
// ===== library types =====

TYPE "mettlerToledoInd560Udt"
   STRUCT
      readMsgSlot : Array[1..4] of Struct
         cmdRespons : Struct
            FP_1 : Bool;
            FP_2 : Bool;
            FP_3 : Bool;
            FP_4 : Bool;
            FP_5 : Bool;
            data_integrity : Bool;
            cmdAck1 : Bool;
            cmdAck2 : Bool;
         END_STRUCT;
         reserved : Byte;   // volt
         data : Real;
         scale_status : Struct
            x08_Enter_Key : Bool;
            x09_Input_1 : Bool;
            x10_Input_2 : Bool;
            x11_Input_3 : Bool;
            x12_Motion : Bool;
            x13_Net_Mode : Bool;
            x14_Data_Integrity_2 : Bool;
            x15_Data_OK : Bool;
            x00_Target_1 : Bool;
            x01_Comparator_1 : Bool;
            x02_Targe_2 : Bool;
            x03_Comparator_2 : Bool;
            x04_Target_3 : Bool;
            x05_Alway_true : Bool;
            x06_TE_bit_1 : Bool;
            x07_TE_bit_2 : Bool;
         END_STRUCT;
      END_STRUCT;
      writeMsgSlot : Array[1..4] of Struct
         cmd : UInt;
         data : Real;
      END_STRUCT;
      run : Struct   // Data calculated from readMsgSlot
         PF : Array[1..4] of USInt;   // Floating point input indication
         cmdAck : Array[1..4] of USInt;
      END_STRUCT;
      occupiedMsgSlots : Array[1..4] of Bool;
      queryDone : Struct
         read : Bool;
         write : Bool;
      END_STRUCT;
   END_STRUCT;
END_TYPE

// folder: Library/Modbus/Core/sb

TYPE "mb_station_block_udt"
   STRUCT
      conf : Struct   // Configuration
         disable : Bool;   // Skip all queries
         read_only : Bool;   // Skip all write queries. (fc 5,6,15,16)
         max_comm_error : USInt := 2;   // Repeating erros before communication_error flag is set
         exec_x_quries : USInt := 1;   // Number of queries to be exec. at each loop.
      END_STRUCT;
      out : Struct   // Outputs
         error : Bool;   // All errors, including communication errors
         error_comm : Bool;   // only communication errors
         finnish : Bool;   // qid is handed over to next device.
      END_STRUCT;
      log : Struct   // Logging for development and debugging.
         connected_time : DTL;   // The time the device was connected to the bus
         disconnected_time : DTL;   // The time, if a device was disconnected to the bus
         done_cnt : UDInt;   // Successfully queries counter for this device
         error_comm_cnt : UDInt;   // Communication erros cnt.
         error_exception_cnt : UDInt;   // Failed queries counter for this device
         error_status : Word;   // Status code from mb_master or mb_client
         error_data_addr : UDInt;   // d_addr for last failed querie; handy for troubleshooting
      END_STRUCT;
      z : Struct   // Internal states.
         header_qid : UInt;   // qid value at device header
         comm_err_cnt : USInt;   // Repeating communication errors
         exec_cnt : USInt;   // Numb. of exec. q. this loop
         offset_qid : UInt := 1;   // Device query id.
         err_hold : Bool;   // Help var for .out.error
      END_STRUCT;
   END_STRUCT;
END_TYPE

// folder: (top level)

FUNCTION_BLOCK "modbus_test"   // FB3, SCL
{ S7_Optimized_Access := 'TRUE' }
VERSION : 0.1
   VAR
      mb_query : "mb_query";
      mb_master_1200_ctrl : "mb_master_1200_ctrl";
      temperature_1 : "Jdrk_RS_WS_N01_8";
      temperature_2 : "Jdrk_RS_WS_N01_8";
      temperature_3 : "Jdrk_RS_WS_N01_8";
      sb_temp_no_answer_1 : "sb_temp_no_anser";
      sb_temp_no_answer_2 : "sb_temp_no_anser";
      sb_temp_no_answer_3 : "sb_temp_no_anser";
      sb_temp_error_1 : "sb_temp_error";
      sb_temp_error_2 : "sb_temp_error";
      sb_temp_error_3 : "sb_temp_error";
   END_VAR
BEGIN
   #mb_master_1200_ctrl.conf.parity := 0;
   #mb_master_1200_ctrl(hardware_id := 263, // "Local~CB_1241_(RS485)",
                        baud := 9600,
                        mb_query := #mb_query);

   #temperature_1(mb_query := #mb_query);
   #temperature_2(mb_query := #mb_query);
   #temperature_3(mb_query := #mb_query);

   #sb_temp_no_answer_1(mb_query := #mb_query);
   #sb_temp_no_answer_2(mb_query := #mb_query);
   #sb_temp_no_answer_3(mb_query := #mb_query);

   #sb_temp_error_1(mb_query := #mb_query);
   #sb_temp_error_2(mb_query := #mb_query);
   #sb_temp_error_3(mb_query := #mb_query);
END_FUNCTION_BLOCK

// folder: Library/Modbus/.Start examples

FUNCTION_BLOCK "modbus_rtu_1200"   // FB3, SCL
{ S7_Optimized_Access := 'TRUE' }
VERSION : 0.1
   VAR
      mb_query : "mb_query";
      mb_master_1200_ctrl : "mb_master_1200_ctrl";
      abb_aquaMaster_device1 : "abb_aquaMaster_3";
      abb_aquaMaster_device2 : "abb_aquaMaster_3";
      abb_aquaMaster_device3 : "abb_aquaMaster_3";
      Auma_valve : "Auma_valve";
      Phoenix_Contact_UPS : "Phoenix_Contact_UPS";
      resault_data_1 : Word;
      Phoenix_Contact_UPS_1 : "Phoenix_Contact_UPS";
   END_VAR
BEGIN
   // hardware_id: Can be found inside "Device configuration".
   // baud:        Bits per sec. (Parity is even by default)
   // timeout:     Automatically calculated if set to T#0s.
   // mb_query:    The FB that connects everything together.
   #mb_master_1200_ctrl(hardware_id := 0, // REPLACE WITH CORRECT ID.
                        baud := 19200,
                        mb_query := #mb_query);

   // Each blocks bellow represent one device on the bus.

   // Three Abb aqua-master's.
   #abb_aquaMaster_device1(mb_addr := 1, mb_query := #mb_query);
   #abb_aquaMaster_device2(mb_addr := 2, mb_query := #mb_query);
   #abb_aquaMaster_device3(mb_addr := 3, mb_query := #mb_query);

   // A valve 
   #Auma_valve(mb_addr := 5, mb_query := #mb_query);


   // A UPS.
   #Phoenix_Contact_UPS(mb_addr := 5, mb_query := #mb_query);

   // A station block can be used both for both modbus rtu and tcp. This
   // is particular useful if a tcp-rtu-gateway is used. The same program
   // could be used, just swap mb_master_1200_ctrl, with mb_client_ctrl.

   // Read holding register 456 from device with modbus address 123.
   // This is an example showing that a query does not necessarily need
   // to be part of a station block (SB) as obove, however making
   // reusable SB's is good practice.
   #mb_query(mb_addr := 123,
             mode := #mb_query.c.read.holding_reg,
             data_addr := 456,
             data_ptr := #resault_data_1);


   // Debugging tip, (no code)
   "mb_Debugging"();
END_FUNCTION_BLOCK

FUNCTION_BLOCK "modbus_rtu_1500"   // FB5, SCL
{ S7_Optimized_Access := 'TRUE' }
VERSION : 0.1
   VAR
      mb_query : "mb_query";
      mb_master_1500_ctrl : "mb_master_1500_ctrl";
      abb_aquaMaster_device1 : "abb_aquaMaster_3";
      abb_aquaMaster_device2 : "abb_aquaMaster_3";
      abb_aquaMaster_device3 : "abb_aquaMaster_3";
      resault_data_1 : Word;
   END_VAR
BEGIN
   // hardware_id:     May be found inside the hardware configuration.
   // operating_mode:  0: RS232, 2: RS422, 4: RS485.
   // baud:            Bits per sec. (Parity is even by default)
   // timeout:         Automatically calculated if set to zero. (T#0s)
   // mb_query:        The FB that connects everything together.
   #mb_master_1500_ctrl(hardware_id := 0, // REPLACE WITH CORRECT ID.
                        operating_mode := 4, // RS-485
                        baud := 19200, // bps
                        mb_query := #mb_query);

   // Each blocks bellow represent one device on the bus. 
   #abb_aquaMaster_device1(mb_addr := 1, mb_query := #mb_query);
   #abb_aquaMaster_device2(mb_addr := 2, mb_query := #mb_query);
   #abb_aquaMaster_device3(mb_addr := 3, mb_query := #mb_query);


   // Debugging tip, (no code)
   "mb_Debugging"();
END_FUNCTION_BLOCK

FUNCTION_BLOCK "modbus_tcp"   // FB79, SCL
{ S7_Optimized_Access := 'TRUE' }
VERSION : 0.1
   VAR
      mb_query : "mb_query";
      mb_client_ctrl : "mb_client_ctrl";
      siemens_PAC3200 : "siemens_PAC3200";
      ip : Array[1..4] of Byte;
      mb_delay_between_queries : "mb_delay_between_queries";
   END_VAR
BEGIN
   // IP-address of the modbus server
   #ip[1] := 192;
   #ip[2] := 168;
   #ip[3] := 1;
   #ip[4] := 2;

   // interface:  Profinet interface.
   //             (Find const. inside "Device configuration")
   // conn_id:    A unique id for each tcp connectin in the plc.
   // ip_addr:    The ip-address of the server. (Array of 4 bytes)
   // tcp_port:   Default port is 502. (UDP isn't available)
   // timeout:    Depends on the network conncetion.
   // mb_query:   The query FB.
   #mb_client_ctrl(interface := 0, // REPLACE WITH CORRECT ID OR CONST,
                                   // Eg. "Local~PROFINET_interface_1",
                   conn_id := 123,
                   ip_addr := #ip,
                   tcp_port := 502,
                   timeout := T#400ms,
                   mb_query := #mb_query);

   #siemens_PAC3200(mb_query := #mb_query);

   // Delay the query execution, this prevent the plc from
   // jamming the network. Adjust the time to your need.
   #mb_delay_between_queries(delay := T#500ms, mb_query := #mb_query);


   // Debugging tip, (no code)
   "mb_Debugging"();
END_FUNCTION_BLOCK

FUNCTION "mb_Readme" : Void   // FC13, SCL
{ S7_Optimized_Access := 'TRUE' }
VERSION : 0.1
BEGIN
   (* Instructions:

   - Add one of the exmple FB's to your PLC.
   - Call that FB from a cyclic OB.
   - Terminate connection to type on the example FB. (Right click the FB)
   - Set hardware_id, buad-rate, ip, tcp-port, etc, to the correct value.
   - Look inside the library and check if there is a ready station block (SB),
     for your program. If there isn't then a new has to be made. 
   - Station blocks can be single-DB's or multi-instances in a FB.
   - Remove the exmple code and example SB's.

   IMPORTANT: As stated above, the start examples fb, need to be terminated 
              from it's type. If the type is edited and later there is a 
              library update, then all the changes will get lost.

   - Instructions need to be of the latest version, 
     this is usually already set:
     * Instructions -> Communication -> Others -> Modbus TCP
     * Instructions -> Communication -> Communication processor -> Modbus
     * Instructions -> Communication -> Communication processor -> Modbus (RTU)  
     * Instructions -> Basic instructions -> Word logic operations -> SEL.
     Change version in the right column.

   *)
END_FUNCTION

// folder: Library/Modbus/.Start examples/Other start examples

FUNCTION_BLOCK "LAD_modbus_rtu"   // FB97, LAD
TITLE = Example modbus rtu
{ S7_Optimized_Access := 'TRUE' }
VERSION : 0.1
// REPLACE hardware_id WITH CORRECT ID.
   VAR
      mb_master_ctrl : "mb_master_1200_ctrl";
      mb_query : "mb_query";
      aquaMaster_device1 : "abb_aquaMaster_3";
      aquaMaster_device2 : "abb_aquaMaster_3";
      Auma_valve : "Auma_valve";
      Phoenix_Contact_UPS : "Phoenix_Contact_UPS";
   END_VAR
   VAR_TEMP   // added for the SCL form of the ladder/FBD networks
      _w1 : Bool;
   END_VAR
BEGIN

REGION Network 1: Modbus master
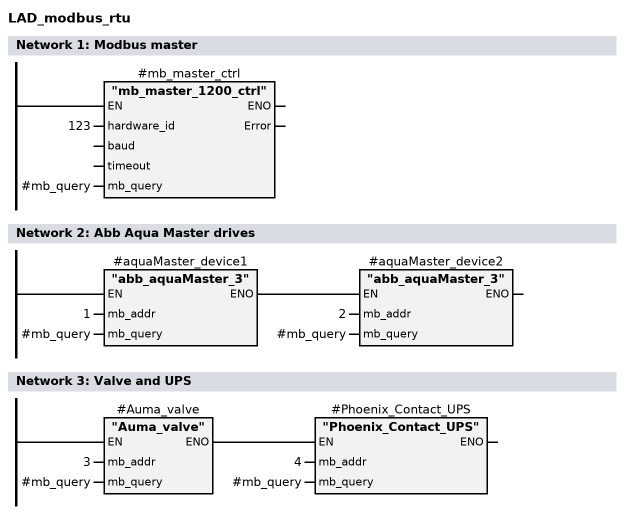
   RUNG wire#powerrail
      #mb_master_ctrl(hardware_id := 123, baud :=, timeout :=, mb_query := #mb_query, Error =>)
   END_RUNG
   // the same network as SCL:
   #mb_master_ctrl(hardware_id := 123, mb_query := #mb_query);   // "mb_master_1200_ctrl"
END_REGION

REGION Network 2: Abb Aqua Master drives
   RUNG wire#powerrail
      #aquaMaster_device1(mb_addr := 1, mb_query := #mb_query)
      #aquaMaster_device2(mb_addr := 2, mb_query := #mb_query)
   END_RUNG
   // the same network as SCL:
   #aquaMaster_device1(mb_addr := 1, mb_query := #mb_query, ENO => #_w1);   // "abb_aquaMaster_3"
   IF #_w1 THEN
       #aquaMaster_device2(mb_addr := 2, mb_query := #mb_query);   // "abb_aquaMaster_3"
   END_IF;
END_REGION

REGION Network 3: Valve and UPS
   RUNG wire#powerrail
      #Auma_valve(mb_addr := 3, mb_query := #mb_query)
      #Phoenix_Contact_UPS(mb_addr := 4, mb_query := #mb_query)
   END_RUNG
   // the same network as SCL:
   #Auma_valve(mb_addr := 3, mb_query := #mb_query, ENO => #_w1);   // "Auma_valve"
   IF #_w1 THEN
       #Phoenix_Contact_UPS(mb_addr := 4, mb_query := #mb_query);   // "Phoenix_Contact_UPS"
   END_IF;
END_REGION
END_FUNCTION_BLOCK

// folder: Library/Modbus/Core

FUNCTION_BLOCK "mb_query"   // FB1, SCL
{ S7_Optimized_Access := 'TRUE' }
VERSION : 0.1
   VAR_INPUT
      mb_addr : UInt;   // Device addr. (0 to 247)
      mode : USInt;   // Function code: 1,2,3,4,5,6,15,16. (siemens mode shifted to 200 - 202)
      data_addr : UDInt;   // Data addr. (raw telegram value, 0-65535)
      data_len : UInt;   // Data len. 0=>Auto detect
   END_VAR
   VAR_OUTPUT
      Done : Bool;   // Successful query
      Error : Bool;   // Failed query
   END_VAR
   VAR_IN_OUT
      data_ptr : Variant;   // Bytes and bools has to add up to whole word(s)
   END_VAR
   VAR
      c : Struct   // Constants
         read : Struct   // Read: 1, 2, 3, 4
            discrete_output : USInt := 101;   // 1 (coils)
            discrete_input : USInt := 102;   // 2
            holding_reg : USInt := 103;   // 3
            input_reg : USInt := 104;   // 4
         END_STRUCT;
         write : Struct   // Write: 5, 6, 15, 16
            single_discrete_output : USInt := 105;   // 5 (coil) (when len. is eq. to 1)
            single_holding_reg : USInt := 106;   // 6 (when len. is eq. to 1)
            discrete_output : USInt := 115;   // 15 (coils)
            holding_reg : USInt := 116;   // 16
         END_STRUCT;
         mode : Struct   // Modicon convention addressing. (Eg: hold.reg. start at 40001)
            read : USInt := 0;   // Mode 0 (fc: 1, 2, 3, 4)
            write_single : USInt := 1;   // Mode 1 (fc: 5, 6) (when len. is eq. to 1)
            write : USInt := 2;   // Mode 2 (fc: 15, 16)
         END_STRUCT;
         auto_len : USInt := 0;   // Length based on data_ptr (Used for data_len)
      END_STRUCT;
      conf : Struct   // Configuration
         buffer_handler : Bool := TRUE;   // enable buffer handler
      END_STRUCT;
      stat : Struct   // Status of last executed query
         done : Bool;   // Successfull
         error : Bool;   // Error, including timeout error
         busy : Bool;   // mb_master or mb_client is busy.
         error_comm : Bool;   // communication error (timeout or bad crc)
         status : Word;   // status word of mb_master or mb_client
      END_STRUCT;
      z : Struct   // Internal states
         q : Struct   // Query params
            mb_addr : UInt := 1;   // Station address
            mode : USInt := 0;   // Function code
            data_addr : UDInt;   // Data address
            data_len : UInt := 0;   // Data length
         END_STRUCT;
         run : Struct   // Constantly changing variables
            qid : UInt := 1;   // query id
            qid_cnt : UInt;   // Query id cnt. increase for each query, reset in controller. One loop each scan
            insert : Bool := TRUE;   // insert query param
            insert2 : Bool;
            write : Bool;   // A write query is inserted
            serialize_err : Int;
         END_STRUCT;
         sb : Struct   // Station block functionality
            sid : UInt;   // Device ID
            sid_cnt : UInt;   // Device id cnt
            sid_retry : UInt := 1;   // Retry device id, qComError
            retry_finished : Bool;
            head_insert : Bool;   // Inc. at mb_query on insert
            head_recive : Bool;   // Inc. at mb_query on rec.
            insert_msg : Bool;   // Stays true even after mb_query has inserted new param.
            reset : Bool;
            log_data_addr : UDInt;   // Tmp.var. for transf. value to mb_device_footer
            log_serialize_err : Int;
         END_STRUCT;
         buffer : Array[0..249] of Byte;
      END_STRUCT;
   END_VAR
   VAR_TEMP
      tLen : UInt;
      tPos : DInt;
      tDiscrete : Bool;
      "e" : Int;
      tBuffer : Array[0..249] of Byte;
   END_VAR
BEGIN
   // Rexhip - Extended modbus library 
   // --------------------------------
   // License:  MIT-license
   // Author:   Ola Bjørnli
   // Web:      www.rexhip.com
   //           github.com/rexhip/rexhip
   //
   // --- --- --- 
   // 
   // mb_query use de-/serialize for data_ptr and hence the function
   // will not work for a discrete queries where the number of bits 
   // dosen't add up to whole bytes. See mb_query_bits.
   //
   // Please read to the documentation and see the examples, before dive
   // into the code bellow, and the rest of the library. (url above)

   REGION Header        
       #Done := #Error := false;

       #z.run.qid_cnt += 1;
       // qid_cnt is increased for every query (above) and reset back to
       // zero in mb_internal_e. Qid (query id) is increased when a query
       // finnish. A query will execute when qit_cnt = qid. Qid is set
       // back to "1" when all queryies has been executed.
       IF #z.run.qid_cnt <> #z.run.qid
           OR #stat.busy // mb_master.busy or mb_client.busy
       THEN
           RETURN;
       END_IF;
   END_REGION

   REGION Auto length
       // data_len=0 => Automatically calculate the length.
       IF #data_len = 0 THEN
           #"e" := Serialize(SRC_VARIABLE := #data_ptr,
                           DEST_ARRAY => #tBuffer,
                           POS := #tPos);
           CASE #mode OF
               101, 102, 105, 115:
                   #tDiscrete := true;
               0..2:
                   CASE #data_addr OF
                       1..9999, 10001..19999:
                           #tDiscrete := true;
                   END_CASE;
           END_CASE;
           #tLen := SEL(G := #tDiscrete,
                        // If "half word", then data_len plus one. 
                        IN0 := DINT_TO_UINT((#tPos + 1) / 2),
                        IN1 := DINT_TO_UINT(#tPos * 8));
       ELSE
           #tLen := #data_len;
       END_IF;
   END_REGION

   REGION Insert and recive
       IF #z.run.insert THEN // Insert query.
           CASE #mode OF
               1, 2, 105, 106, 115, 116: // Write  
                   #z.run.write := true;
               ELSE // Read
                   #z.run.write := false;
           END_CASE;
           // The params is transfered over to the udt. They are later
           // transfered from the udt to mb_master or mb_client.
           #z.q.mb_addr := #mb_addr;
           #z.q.mode := #mode;
           #z.q.data_addr := #data_addr;
           #z.q.data_len := #tLen;

           // Reset var for this query. #e will be zero if no error for
           // auto_len above. A value different from zero means a error.
           #z.run.serialize_err := #"e";

           IF #conf.buffer_handler AND #z.run.write THEN
               // Copy the content of #data_ptr to the buffer.
               #tPos := 0; // Start at the beginning of the buffer.
               #z.run.serialize_err := // Zero if no error.
               Serialize(SRC_VARIABLE := #data_ptr,
                         DEST_ARRAY => #z.buffer,
                         POS := #tPos);
           END_IF;
           // False while waiting for the resualt.
           #z.run.insert := false;
           // insert2 make sure that a query is only exec. once. 
           // Don't execute if serialize error. 0 => no error
           #z.run.insert2 := #z.run.serialize_err = 0;
           // A msg. to station block foother FC, a new query has
           // been inserted.
           #z.sb.head_insert := true;

           // If the query is finnished. (with or without error)  
       ELSIF #stat.done OR #stat.error THEN

           // Make sure that the query resault really belong to this
           // query. This can be false if an other query before is
           // surrounded by a if-statement
           IF #z.q.mb_addr = #mb_addr
               AND #z.q.mode = #mode
               AND #z.q.data_addr = #data_addr
               AND #z.q.data_len = #tLen
           THEN
               IF #stat.done // Successfull query (no error)
                   AND NOT #z.run.write  // If it's a read query
                   AND #conf.buffer_handler
               THEN
                   // Copy the content from the buffer to #data_ptr
                   #tPos := 0; // Start at the beginning of the buffer.
                   #z.run.serialize_err := // Zero if no error.
                   Deserialize(SRC_ARRAY := #z.buffer,
                               DEST_VARIABLE => #data_ptr,
                               POS := #tPos);
               END_IF;
               #Done := #stat.done AND #z.run.serialize_err = 0;
               #Error := NOT #Done;

               // Temperary store value, so it can be picked up in the
               // sb footer.
               #z.sb.log_data_addr := #data_addr;
               #z.sb.log_serialize_err := #z.run.serialize_err;
               // Msg. to mb_station_footer.
               #z.sb.head_recive := true;
           END_IF;
           #z.run.qid += 1; // Move on to next query
           #z.run.insert := true; // Prepare for the next query.
       END_IF;
   END_REGION
END_FUNCTION_BLOCK

// folder: Library/Modbus/Core/Ctrl

FUNCTION_BLOCK "mb_client_ctrl"   // FB9, SCL
{ S7_Optimized_Access := 'TRUE' }
VERSION : 1.0
   VAR_INPUT
      interface : Hw_Any := 64;   // Profinet interface id
      conn_id : Conn_Ouc := 123;   // Connection id
      ip_addr : Array[1..4] of Byte;   // IPv4
      tcp_port : UInt := 502;   // TCP port
      timeout : Time := T#1S;
   END_VAR
   VAR_OUTPUT
      Error : Bool;   // error flag with tof timer
   END_VAR
   VAR_IN_OUT
      mb_query : "mb_query";   // udt mb
   END_VAR
   VAR
      conf : Struct
         disconnect : Bool := FALSE;
         retries : USInt := 0;
      END_STRUCT;
      client : MB_CLIENT;
      tcon_ip_v4 : TCON_IP_v4;
      ton_timeout : TON_TIME;
      ton_timeout_q : Bool;
      timeout_state : SInt;
      tdiscon : TDISCON;
      tdiscon_bool : Bool;
      end : "mb_internal_e";
   END_VAR
BEGIN
   // Rexhip - Extended modbus library.
   // Please see top section of mb_query for more info.
   // 
   // Please read the documentation, before dive into the code bellow

   // For use with modbus tcp.

   #tcon_ip_v4.InterfaceId := #interface;
   #tcon_ip_v4.ID := #conn_id;
   #tcon_ip_v4.ConnectionType := 11; // tcp
   #tcon_ip_v4.ActiveEstablished := true;
   #tcon_ip_v4.RemoteAddress.ADDR := #ip_addr;
   #tcon_ip_v4.RemotePort := #tcp_port;

   // If mb_client does not establish a connection it will not
   // throw timeout error. Timeout is handled manually for that
   // case. 16#7002: Intermediate call. Connection is being
   // established.
   #ton_timeout(IN := #client.STATUS = 16#7002,
                PT := #timeout,
                Q => #ton_timeout_q);

   IF #mb_query.z.run.insert2 THEN
       #mb_query.z.run.insert2 := false;
       // After query has been exec. data_len will be set to zero.
       // This will make sure that a query is not executed twice,
       // becouse data_len = 0, will generate a error.
       #client.MB_DATA_LEN := #mb_query.z.q.data_len;
   END_IF;

   #client.MB_Unit_ID := UINT_TO_BYTE(#mb_query.z.q.mb_addr);
   #client.Rcv_Timeout :=
   UDINT_TO_REAL(T_CONV(#timeout)) * 0.001; // In secounds
   #client.Retries := #conf.retries;
   #client(REQ := NOT #client.BUSY
           AND NOT #mb_query.z.run.insert
           AND NOT #client.DISCONNECT
           AND #mb_query.z.run.qid <> 0,
           DISCONNECT := #conf.disconnect
           OR #tdiscon.BUSY
           OR #timeout_state = 1,
           MB_MODE := #mb_query.z.q.mode,
           MB_DATA_ADDR := #mb_query.z.q.data_addr,
           MB_DATA_LEN := #client.MB_DATA_LEN,
           BUSY => #mb_query.stat.busy,
           DONE => #mb_query.stat.done,
           ERROR => #mb_query.stat.error,
           STATUS => #mb_query.stat.status,
           MB_DATA_PTR := #mb_query.z.buffer,
           CONNECT := #tcon_ip_v4);

   IF #client.DONE OR #client.ERROR THEN
       // Make sure that a query is not exec. twice.
       IF #client.MB_DATA_LEN <> 0 THEN
           #mb_query.z.q.data_len := #client.MB_DATA_LEN;
           #client.MB_DATA_LEN := 0;
           // A secound exec. will cause a error code when
           // data_len is set to zero.
       END_IF;

       // Timeout handeling.
       #mb_query.stat.error_comm := #mb_query.stat.error
       // blocked_proc_timeout or rcv_timeout
       AND (#mb_query.stat.status = 16#818C
       // No response from the server
       OR #mb_query.stat.status = 16#80C8
       OR #timeout_state = 2); // Reconnect after disconnect.

       #timeout_state := 0; // Reset
   ELSE
       CASE #timeout_state OF
           0: // Normal opperation (no ton_timeout)
               #timeout_state := BOOL_TO_SINT(#ton_timeout_q);
           1: // Disconnect and reconnect mb_client.
               #timeout_state := 2;
       END_CASE;
   END_IF;

   // If a new download has taken place, and this block is
   // re-initialize, then the mb_client block will output the
   // error code saying that: "Attempt being made to
   // re-establish an existing connection." (16#80A3). The
   // solution to this problem is to disconnect and then
   // reconnect.
   #tdiscon(REQ := #client.STATUS = 16#80A3, ID := #conn_id);

   // End is comman for both tcp and rtu.
   #end(mb_query := #mb_query, Error => #Error);
END_FUNCTION_BLOCK

FUNCTION_BLOCK "mb_master_1500_ctrl"   // FB10, SCL
{ S7_Optimized_Access := 'TRUE' }
VERSION : 1.0
   VAR_INPUT
      hardware_id : Port;   // hardware id
      operating_mode : USInt := 4;   // 0: RS232, 2: RS422, 4: RS485.
      baud : UDInt := 19200;   // Bits per sec.
      timeout : Time;   // Automatically calculated if set to zero. (T#0s)
   END_VAR
   VAR_OUTPUT
      Error : Bool;   // One or more errors in the whole application.
   END_VAR
   VAR_IN_OUT
      mb_query : "mb_query";
   END_VAR
   VAR
      conf : Struct
         parity : UInt := 2;   // 0=no-parity, 1=odd, 2=even.
         retries : USInt := 0;
      END_STRUCT;
      comm_load : Modbus_Comm_Load;
      master : Modbus_Master;
      buffer : "mb_internal_b";
      end : "mb_internal_e";
      comm_load_done : Bool;
   END_VAR
BEGIN
   // Rexhip - Extended modbus library.
   // Please see top section of mb_query for more info.
   //
   // RTU master for S7-1500
   // 
   // This master blocks works for both S7-1200 and S7-1500.
   // For S7-1200 it's recommended to use the other master 
   // block mb_master_1200_ctrl, because it use less memory.
   // Please read the documentation, before dive into the
   // code bellow


   // master header
   "mb_internal_h"(mode104 := true,
                   timeout := #timeout,
                   baud := #baud,
                   resp_to := #comm_load.RESP_TO,
                   mode := #master.MODE,
                   data_addr := #master.DATA_ADDR,
                   data_len := #master.DATA_LEN,
                   buffer := #buffer,
                   mb_query := #mb_query);

   // Initiate the hardware.
   #comm_load.RETRIES := #conf.retries;
   #comm_load.MODE := #operating_mode;
   #comm_load(REQ := NOT #comm_load_done,
              PORT := #hardware_id,
              BAUD := #baud,
              PARITY := #conf.parity,
              RESP_TO := #comm_load.RESP_TO,
              MB_DB := #master.MB_DB);
   IF #comm_load.DONE THEN
       #comm_load_done := true;
   ELSIF #comm_load.ERROR THEN
       #comm_load_done := false;
   END_IF;

   // The core master block.
   #master(REQ := #comm_load_done
           AND NOT #master.BUSY
           AND NOT #mb_query.z.run.insert
           AND #mb_query.z.run.qid <> 0,
           MB_ADDR := #mb_query.z.q.mb_addr,
           MODE := #master.MODE,
           DATA_ADDR := #master.DATA_ADDR,
           DATA_LEN := #master.DATA_LEN,
           DONE => #mb_query.stat.done,
           BUSY => #mb_query.stat.busy,
           STATUS => #mb_query.stat.status,
           DATA_PTR := #buffer.buffer);
   #mb_query.stat.error := #master.ERROR OR #comm_load.ERROR;

   // master footer
   "mb_internal_f"(data_len := #master.DATA_LEN,
                   buffer := #buffer,
                   mb_query := #mb_query);

   // End is comman for both tcp and rtu.
   #end(mb_query := #mb_query,
        Error => #Error);
END_FUNCTION_BLOCK

FUNCTION_BLOCK "mb_master_1200_ctrl"   // FB90, SCL
{ S7_Optimized_Access := 'TRUE' }
VERSION : 1.0
   VAR_INPUT
      hardware_id : Port := 0;   // Hardware id
      baud : UDInt := 19200;   // Bits per second
      timeout : Time;   // Automatically calculated if set to zero. (T#0s)
   END_VAR
   VAR_OUTPUT
      Error : Bool;   // One or more errors in the whole application.
   END_VAR
   VAR_IN_OUT
      mb_query : "mb_query";
   END_VAR
   VAR
      conf : Struct
         parity : UInt := 2;   // 0=no-parity, 1=odd, 2=even.
         retries : USInt := 0;
      END_STRUCT;
      comm_load : MB_COMM_LOAD;
      master : MB_MASTER;
      buffer : "mb_internal_b";
      end : "mb_internal_e";
   END_VAR
   VAR_TEMP
      tmp_err : Bool;
   END_VAR
BEGIN
   // Rexhip - Extended modbus library.
   // Please see top section of mb_query for more info.
   // 
   // RTU master for S7-1200
   // 
   // This FB use less memory then mb_master_1500_ctrl, but it
   // only works for S7-1200 PLC's. Please read the
   // documentation, before dive into the code bellow

   // Master header
   "mb_internal_h"(mode104 := false,
                   timeout := #timeout,
                   baud := #baud,
                   resp_to := #comm_load.RESP_TO,
                   mode := #master.MODE,
                   data_addr := #master.DATA_ADDR,
                   data_len := #master.DATA_LEN,
                   buffer := #buffer,
                   mb_query := #mb_query);

   // Initiate the hardware
   #comm_load.RETRIES := #conf.retries;
   #comm_load(REQ := NOT #comm_load.DONE,
              PORT := #hardware_id,
              BAUD := #baud,
              PARITY := #conf.parity,
              RESP_TO := #comm_load.RESP_TO,
              MB_DB := #master);

   // The core master block.
   #master(REQ := #comm_load.DONE
           AND NOT #master.BUSY
           AND NOT #mb_query.z.run.insert
           AND #mb_query.z.run.qid <> 0,
           MB_ADDR := #mb_query.z.q.mb_addr,
           MODE := #master.MODE,
           DATA_ADDR := #master.DATA_ADDR,
           DATA_LEN := #master.DATA_LEN,
           DONE => #mb_query.stat.done,
           BUSY => #mb_query.stat.busy,
           STATUS => #mb_query.stat.status,
           DATA_PTR := #buffer.buffer);
   #mb_query.stat.error := #master.ERROR OR #comm_load.ERROR;

   // Master footer
   "mb_internal_f"(data_len := #master.DATA_LEN,
                   buffer := #buffer,
                   mb_query := #mb_query);

   // End is comman for both tcp and rtu.
   #end(mb_query := #mb_query,
        Error => #Error);
END_FUNCTION_BLOCK

// folder: Library/Modbus/Core/Internal

FUNCTION_BLOCK "mb_internal_b"   // FB6, SCL
{ S7_Optimized_Access := 'FALSE' }
VERSION : 0.1
   VAR
      buffer : Array[0..249] of Byte;
   END_VAR
BEGIN
   (*
   - Buffer for mb_master. (modbus rtu)
   - This block has optimize data access disabled.
   - For RTU, please do not delete the even there is no code bellow.
   - This block isn't needed for modbus tcp.
   *)
END_FUNCTION_BLOCK

FUNCTION_BLOCK "mb_internal_e"   // FB7, SCL
{ S7_Optimized_Access := 'TRUE' }
VERSION : 0.1
   VAR_OUTPUT
      Error : Bool;
   END_VAR
   VAR_IN_OUT
      mb_query : "mb_query";
   END_VAR
   VAR
      err_hold : Bool;
   END_VAR
BEGIN
   // Internal function - common for both rtu and tcp.

   // insert_msg is only written here, while insert will be 
   // changed inside the queries.
   #mb_query.z.sb.insert_msg := #mb_query.z.run.insert;

   // Anti wind up effect for qid. msg. to devices that they should
   // reset if qid grow bigger then 60000. (See mb_station_block_header)
   #mb_query.z.sb.reset := false;
   IF #mb_query.z.run.qid > 60000 THEN
       #mb_query.z.sb.reset := true;
   END_IF;

   // #error will be keeped true as long there is at least one query that
   // generate a error. 
   IF #mb_query.stat.error THEN
       #Error := true;
       #err_hold := true;
   END_IF;

   // If all queries has been executed,
   IF #mb_query.z.run.qid > #mb_query.z.run.qid_cnt THEN

       // Error handeling (see above)
       IF NOT #err_hold THEN
           #Error := false;
       END_IF;
       #err_hold := false;

       // Start over again on the first query.
       #mb_query.z.run.qid := 1;

       // The retry-id is the device that get to have retry to restoring
       // communication after the error_comm flag is set for the station.
       // When one query loop has occurred the retry id is incremented. 
       #mb_query.z.sb.sid_retry := #mb_query.z.sb.sid_retry + 1;

       // retry_finished is set after one retry has taken place. 
       // The station that has the retry-token only has one try to make 
       // successfully query.
       #mb_query.z.sb.retry_finished := false;
       IF #mb_query.z.sb.sid_retry > #mb_query.z.sb.sid_cnt THEN
           #mb_query.z.sb.sid_retry := 1;
       END_IF;

       // Station id: (not in use)
       #mb_query.z.sb.sid := #mb_query.z.sb.sid + 1;
       IF #mb_query.z.sb.sid > #mb_query.z.sb.sid_cnt THEN
           #mb_query.z.sb.sid := 1;
       END_IF;
   END_IF;

   #mb_query.z.run.qid_cnt := 0; // (Incremented in mb_query)
   #mb_query.z.sb.sid_cnt := 0; // (Incremented in mb_station_block_header)
END_FUNCTION_BLOCK

FUNCTION "mb_internal_f" : Void   // FC2, SCL
{ S7_Optimized_Access := 'TRUE' }
VERSION : 0.1
   VAR_IN_OUT
      data_len : UInt;
      buffer : "mb_internal_b";
      mb_query : "mb_query";
   END_VAR
   VAR_TEMP
      comm_error : Bool;
   END_VAR
BEGIN
   // Internal function - master footer

   IF #mb_query.stat.done OR #mb_query.stat.error THEN
       // Make sure that a query isn't exec. twice.
       IF #data_len <> 0 THEN
           #mb_query.z.q.data_len := #data_len;
           #data_len := 0;
       END_IF;

       IF NOT #mb_query.z.run.write THEN // A read query.
           #mb_query.z.buffer := #buffer.buffer;
       END_IF;

       // Communication error (Handled different from other errors)
       CASE WORD_TO_UINT(#mb_query.stat.status) OF
           16#80C8, // Timeout
           16#8380, // Bad CRC 
           16#80E1, // Parity error
           16#80E2: // Framing error
               #comm_error := true;
       END_CASE;
   END_IF;

   #mb_query.stat.error_comm := #mb_query.stat.error AND #comm_error;
END_FUNCTION

FUNCTION "mb_internal_h" : Void   // FC4, SCL
{ S7_Optimized_Access := 'TRUE' }
VERSION : 0.1
   VAR_INPUT
      mode104 : Bool;
      timeout : Time;
      baud : UDInt;
   END_VAR
   VAR_IN_OUT
      resp_to : UInt;
      mode : USInt;
      data_addr : UDInt;
      data_len : UInt;
      buffer : "mb_internal_b";
      mb_query : "mb_query";
   END_VAR
BEGIN
   // Internal function - master header

   IF #mb_query.z.run.insert2 THEN
       #mb_query.z.run.insert2 := false;
       #mode := 0;
       #data_len := #mb_query.z.q.data_len;
       // mb_master use modicon convention address.
       CASE #mb_query.z.q.mode OF
           0..2: // Read and write
               #mode := #mb_query.z.q.mode;
               #data_addr := #mb_query.z.q.data_addr;
           101:  // Read output bits
               #data_addr := 1 + #mb_query.z.q.data_addr;
           102:  // Read input bits
               #data_addr := 10001 + #mb_query.z.q.data_addr;
           103:  // Read holding reg.
               #data_addr := 400001 + #mb_query.z.q.data_addr;
           104:  // Read input word
               IF #mode104 THEN
                   #mode := 104;
                   #data_addr := #mb_query.z.q.data_addr;
               ELSE
                   #data_addr := 30001 + #mb_query.z.q.data_addr;
               END_IF;
           105:  // Writing a single output bit
               #mode := 1;
               #data_addr := 1 + #mb_query.z.q.data_addr;
           106:  // Writing a single holding register
               #mode := 1;
               #data_addr := 400001 + #mb_query.z.q.data_addr;
           115: // Writing multiple output bits
               #mode := 2;
               #data_addr := 1 + #mb_query.z.q.data_addr;
           116: // Writing multiple holding registers
               #mode := 2;
               #data_addr := 400001 + #mb_query.z.q.data_addr;
           ELSE
               #mode := #mb_query.z.q.mode;
               #data_addr := #mb_query.z.q.data_addr;
       END_CASE;

       IF #mb_query.z.run.write THEN
           #buffer.buffer := #mb_query.z.buffer;
       END_IF;
   END_IF;

   // Automatically adjust timeout.
   #resp_to := SEL(G := #timeout = T#0s,
                   IN0 := T_CONV(#timeout),
                   IN1 := UDINT_TO_UINT(3200000 / #baud));
END_FUNCTION

// folder: Library/Modbus/Core/Special

FUNCTION_BLOCK "mb_delay"   // FB11, SCL
{ S7_Optimized_Access := 'TRUE' }
VERSION : 0.1
   VAR_INPUT
      delay : Time;
   END_VAR
   VAR_IN_OUT
      mb_query : "mb_query";
   END_VAR
   VAR
      "timer" : TON_TIME;
      qid : UInt := 1;
      wait : Bool;
   END_VAR
BEGIN
   // For use with modbus tcp, so the client dosen't jam a network.
   // The function halt execution of queries for a certain time

   #mb_query.z.run.qid_cnt += 1;  // The timer occupy one qid.

   IF #wait THEN // If the timer has been activated.
       #"timer"(IN := true,
              PT := #delay);
       IF #"timer".Q THEN
           #mb_query.z.run.qid := #qid + 1;
           RESET_TIMER(#"timer");
           #wait := false;
       END_IF;
   ELSIF #mb_query.z.run.qid_cnt = #mb_query.z.run.qid
       AND NOT #mb_query.stat.busy
   THEN
       #qid := #mb_query.z.run.qid; // Store the value
       #mb_query.z.run.qid := 0; // Stop exec.
       #wait := true;
   END_IF;
END_FUNCTION_BLOCK

FUNCTION_BLOCK "mb_delay_between_queries"   // FB13, SCL
{ S7_Optimized_Access := 'TRUE' }
VERSION : 0.1
   VAR_INPUT
      delay : Time;
   END_VAR
   VAR_IN_OUT
      mb_query : "mb_query";
   END_VAR
   VAR
      "timer" : IEC_TIMER;
      wait : Bool;
      qid : UInt := 1;
   END_VAR
BEGIN
   // For use with modbus tcp, so the client dosen't jam a network.
   // The function halt execution of queries for a certain time
   // not just once, but between every query.  

   IF #wait THEN
       #"timer".TON(IN := true,
                  PT := #delay);
       IF #"timer".Q THEN
           #mb_query.z.run.qid := #qid;
           RESET_TIMER(#"timer");
           #wait := false;
       END_IF;
   ELSIF #mb_query.z.run.qid <> #qid
       AND #mb_query.z.run.qid <> 0
       AND NOT #mb_query.stat.busy
   THEN
       #qid := #mb_query.z.run.qid;
       #mb_query.z.run.qid := 0; // Stop the "loop"
       #wait := true;
   END_IF;
END_FUNCTION_BLOCK

FUNCTION "mb_dataptr_eq_buffer" : Bool   // FC3, SCL
{ S7_Optimized_Access := 'TRUE' }
VERSION : 0.1
   VAR_IN_OUT
      data_ptr : Variant;
      mb_query : "mb_query";
   END_VAR
   VAR_TEMP
      tmp_buffer : Array[0..249] of Byte;
      pos : DInt;
      c : Int;
      "e" : Int;
   END_VAR
BEGIN
   // Most use cases will not need this function !
   // Example:
   // 
   // #mb_query(mb_addr := 123,
   //           mode := #mb_query.c.write.holding_reg,
   //           data_addr := 456,
   //           data_ptr := #data);
   //
   // IF #mb_query.Done AND
   //     "mb_dataPtr_eq_buffer"(data_ptr := #data, mb_query := #mb_query)
   // THEN
   //      // If there are for some reason two write queries that has exatly
   //      // the same parameters, then the Done-flag may not be enough to
   //      // determine which query has been executed. To compare data as
   //      // well, data_ptr to the buffer, then this use this function. It
   //      // will return true if the content is the same.
   // END_IF;
   //
   // ------- 

   #mb_dataptr_eq_buffer := true; // Init. value

   #"e" := Serialize(SRC_VARIABLE := #data_ptr,
                   DEST_ARRAY => #tmp_buffer,
                   POS := #pos);

   // Looking for differences.
   FOR #c := 0 TO #pos - 1 DO
       IF #tmp_buffer[#c] <> #mb_query.z.buffer[#c] THEN
           #mb_dataptr_eq_buffer := false;
           EXIT;
       END_IF;
   END_FOR;
END_FUNCTION

FUNCTION "mb_query_bits" : Void   // FC9, SCL
{ S7_Optimized_Access := 'TRUE' }
VERSION : 0.1
   VAR_IN_OUT
      data_ptr : Array[*] of Bool;
      mb_query : "mb_query";
   END_VAR
   VAR_TEMP
      discrete : Bool;
      dommy : Bool;
      lower : DInt;
      upper : DInt;
      bits : UInt;
      bytes : UDInt;   // bytes
   END_VAR
BEGIN
   // This function should be used when the number of bits dosen't
   // add up to whole bytes, for function codes: 1, 2, 5 and 15. 
   // 
   // data_ptr need to be a one dimensional array of bools.
   // --- --- ---

   IF #mb_query.z.run.qid_cnt + 1 <> #mb_query.z.run.qid
       OR #mb_query.stat.busy
   THEN
       // Skip query, qid will not match qid_cnt and
       // my_query will return.
       #mb_query(data_ptr := #dommy);
       RETURN;
   END_IF;

   // Some preparing calculations.
   CASE #mb_query.mode OF // A discrete query ?
       101, 102, 105, 115:
           #discrete := true;
       0..2:
           CASE #mb_query.data_addr OF
               1..9999, 10001..19999:
                   #discrete := true;
           END_CASE;
   END_CASE;
   #lower := LOWER_BOUND(ARR := #data_ptr, DIM := 1);
   #upper := UPPER_BOUND(ARR := #data_ptr, DIM := 1);
   #bits := DINT_TO_UINT(#upper - #lower + 1); // Elements in array.

   // Auto data len ?
   IF #mb_query.data_len = #mb_query.c.auto_len THEN
       #bytes := (#bits + 7) / 8; // CEIL()
       #mb_query.data_len := SEL(G := #discrete,
                                 IN0 := (#bits + 15) / 16, // CEIL()
                                 IN1 := #bits);
   ELSE
       #bytes := SEL(G := #discrete,
                     IN0 := #mb_query.data_len * 2, // 1 word -> 2 bytes
                     IN1 := (#mb_query.data_len + 7) / 8); // CEIL()
   END_IF;

   // Insert query.
   IF #mb_query.z.run.insert THEN
       CASE #mb_query.mode OF
           1, 2, 105, 106, 115, 116: // A write query.
               // Copy the content from data_ptr to the buffer.
               GATHER_BLK(IN := #data_ptr[#lower],
                          COUNT_OUT := #bytes,
                          OUT => #mb_query.z.buffer[0]);
       END_CASE;
   END_IF;

   // Disable buf.h. inside mb_query.
   #mb_query.conf.buffer_handler := false;

   // Run the query.
   #mb_query(data_ptr := #dommy);

   #mb_query.conf.buffer_handler := true; // Enable buf.h. again.
   #mb_query.data_len := #mb_query.c.auto_len; // Back to auto.

   // Handle resualt.
   IF #mb_query.Done // The query above.
       AND NOT #mb_query.z.run.write  // A read query
   THEN
       // Copy the content from the buffer to data_ptr.
       SCATTER_BLK(IN := #mb_query.z.buffer[0],
                   COUNT_IN := #bytes,
                   OUT => #data_ptr[#lower]);
   END_IF;
END_FUNCTION

FUNCTION "mb_execute" : Bool   // FC12, SCL
{ S7_Optimized_Access := 'TRUE' }
VERSION : 0.1
   VAR_IN_OUT
      mb_query : "mb_query";
   END_VAR
   VAR_TEMP
      dommy : Bool;
   END_VAR
BEGIN
   // Most use cases will not need this function !
   // Example:
   // 
   // IF "mb_execute"(#mb_query) THEN
   //     
   //     // Preparing calculations.
   //     
   //     #mb_query(data_addr := 2, data_ptr := #data);
   // END_IF;
   //
   // Usefull if some CPU demanding calculation need to be done
   // before a write query is inserted. Note that a query can later
   // be aborted, thought mb_execute return true.

   #mb_execute := #mb_query.z.run.qid_cnt + 1 = #mb_query.z.run.qid
   (* *)AND NOT #mb_query.stat.busy;

   IF NOT #mb_execute THEN
       #mb_query(data_ptr := #dommy);
   END_IF;
END_FUNCTION

// folder: Library/Modbus/Core/Special/Special code snippets examples

FUNCTION_BLOCK "Example Done and error"   // FB56, SCL
{ S7_Optimized_Access := 'TRUE' }
VERSION : 0.1
   VAR_IN_OUT
      mb_query : "mb_query";
   END_VAR
   VAR
      query1_data : Word;
      done_cnt : UInt;
      query2_data : Word;
   END_VAR
BEGIN
   // To get information about when a particular query has executed.

   #mb_query(mb_addr := 123,
             mode := #mb_query.c.write.holding_reg,
             data_addr := 456,
             data_ptr := #query1_data);

   // The if-statement bellow has to be put after the particular 
   // query, and before the next query.    

   IF #mb_query.Done THEN
       // Some action after a successfully query.    
       #done_cnt += 1; // Eg. count successfully queries.

   ELSIF #mb_query.Error THEN
       // Some action if a faild query.    

       // #mb_query.stat.status , gives more information about 
       // the error.         

       IF #mb_query.stat.error_comm THEN
           ; // Some particular action if communication error.
       END_IF;

   END_IF;

   // Next query...
   #mb_query(mb_addr := 111,
             mode := #mb_query.c.read.holding_reg,
             data_addr := 789,
             data_ptr := #query2_data);
END_FUNCTION_BLOCK

FUNCTION_BLOCK "Example Swap"   // FB78, SCL
{ S7_Optimized_Access := 'TRUE' }
VERSION : 0.1
   VAR_IN_OUT
      mb_query : "mb_query";
   END_VAR
   VAR
      static_tmp_var : Word;
      value : Word;
   END_VAR
BEGIN
   // For some modbus devices, when two registers are combined into one,
   // the data is stored as little endian, not big endian like Siemens 
   // PLC does. To solve this, the SWAP function needs to be utilized.
   #mb_query(mb_addr := 123,
             mode := #mb_query.c.read.holding_reg,
             data_addr := 123,
             data_ptr := #static_tmp_var);

   #value := SWAP(#static_tmp_var);


   // For other device, when two registers are combined, the least significant 
   // word is stored first and the most significant word is stored in the 
   // following register. When this is the case, the ROR-function needs 
   // to be used.
   #mb_query(mb_addr := 123,
             mode := #mb_query.c.read.holding_reg,
             data_addr := 123,
             data_ptr := #static_tmp_var);

   #value := ROR(IN := #static_tmp_var, N := 16);


   // In some situation both SWAP and ROR need to be used.
   #mb_query(mb_addr := 123,
             mode := #mb_query.c.read.holding_reg,
             data_addr := 123,
             data_ptr := #static_tmp_var);

   #value := SWAP(ROR(IN := #static_tmp_var, N := 16));

   // How the data is stored, is usually described in the
   // data sheet of each device.
END_FUNCTION_BLOCK

FUNCTION_BLOCK "Example Read first"   // FB85, SCL
{ S7_Optimized_Access := 'TRUE' }
VERSION : 0.1
   VAR_INPUT
      input1 : Bool;
      input2 : Bool;
   END_VAR
   VAR_IN_OUT
      mb_query : "mb_query";
   END_VAR
   VAR
      write : Bool;
      data : Word;
   END_VAR
BEGIN
   // Sometimes only some bits in a word need to be manipulated, 
   // without touching the other bits, bellow is an example how 
   // that can be achieved.

   #mb_query.mb_addr := 123;
   #mb_query.data_addr := 456;

   IF #write THEN // (Initially false)

       // Manipulating only bit 5 and 11
       #data.%X5 := #input1;
       #data.%X11 := #input2;

       #mb_query(mode := #mb_query.c.write.holding_reg,
                 data_ptr := #data);

   ELSE // read the register before write to the same one.
       #mb_query(mode := #mb_query.c.read.holding_reg,
                 data_ptr := #data);

       // Has query above been executed successfully?
       IF #mb_query.Done THEN
           #write := true;
       END_IF;

   END_IF;
END_FUNCTION_BLOCK

FUNCTION_BLOCK "Example Forced execution order"   // FB89, SCL
{ S7_Optimized_Access := 'TRUE' }
VERSION : 0.1
   VAR_IN_OUT
      mb_query : "mb_query";
   END_VAR
   VAR
      state : Int;
      query_1 : Word;
      query_2 : UInt;
      query_3 : Word;
      query_4 : Word;
   END_VAR
BEGIN
   // If the execution need to be forced to a given order, then the 
   // example bellow can be followed.

   CASE #state OF

       0:  // 1st query
           #mb_query(mb_addr := 123,
                     mode := #mb_query.c.write.holding_reg,
                     data_addr := 123,
                     data_ptr := #query_1);
           #state += BOOL_TO_SINT(#mb_query.Done);
           // «#mb_query.done» is set true when the query above is done 
           // successfully. When next query is executed, «#mb_query.done»
           // is set back false.

       1:  // 2nd query
           #mb_query(mb_addr := 123,
                     mode := #mb_query.c.write.holding_reg,
                     data_addr := 456,
                     data_ptr := #query_2);
           #state += BOOL_TO_SINT(#mb_query.Done);

       2:  // 3rd query
           #mb_query(mb_addr := 123,
                     mode := #mb_query.c.read.holding_reg,
                     data_addr := 789,
                     data_ptr := #query_3);
           IF #mb_query.Done THEN
               #state := 0;
           END_IF;
   END_CASE;

   // 4th query, this query is executed three times as often 
   // as the queries above.
   #mb_query(mb_addr := 123,
             mode := #mb_query.c.read.input_reg,
             data_addr := 1234,
             data_ptr := #query_4);
END_FUNCTION_BLOCK

// folder: Library/Modbus/Core/sb

FUNCTION "mb_station_block_header" : Void   // FC10, SCL
{ S7_Optimized_Access := 'TRUE' }
VERSION : 1.0
   VAR_IN_OUT
      sb : "mb_station_block_udt";
      mb_query : "mb_query";
   END_VAR
BEGIN
   // Rexhip - Extended modbus library.
   // Read the top section of mb_query for more documentation.

   #mb_query.data_len := 0; // Default is auto-length.
   #mb_query.conf.buffer_handler := true;

   // If device blocks are executeded in diffrent order, a wide wind
   // up effect will occur, (in same OB) this will prevent that.
   IF #mb_query.z.sb.reset THEN
       #sb.z.header_qid := #mb_query.z.run.qid_cnt + 1;
   END_IF;

   // Device id cnt. The first device has id "1". Increased in every
   // mb_device_header, reseted in mb_client_ctrl or mb_master_ctrl.
   #mb_query.z.sb.sid_cnt += 1;

   // mb_query set the same bellow variables to true, at insert or recive.
   // This informastion is later used at the footer.
   #mb_query.z.sb.head_insert := false;
   #mb_query.z.sb.head_recive := false;

   // Reset order, a variable that makes queries in a sb execute in order.
   // #mb_query.z.sb.order := false;

   // When #mb.mb.q.qid = #mb.mb.run.qid_cnt => "This" device has the
   // query-token !
   // - If the query-token points at this device header, or it point to a
   //   query in the previous device, that is surrounded by a if-statement
   //   and the statement is now false.
   // - A gid change can only be done if not "busy", this is to avoid a
   //   resualt from one query being intercepted by another
   IF #mb_query.z.run.qid > #mb_query.z.run.qid_cnt
       AND #mb_query.z.run.qid <= #sb.z.header_qid
       AND NOT #mb_query.stat.busy
   THEN
       // Reset.
       #mb_query.z.run.insert := true;

       // At first the offset_qid points at the first query of this
       // device. When it has executed the offset will point at the
       // second query. When all queries has executed the offset will
       // be reset back to the first query. (footer) 
       #mb_query.z.run.qid :=
       #sb.z.header_qid + #sb.z.offset_qid;

       // Order is a variable that makes queries in sb execute in order.
       //    #mb_query.z.sb.order := true;
   END_IF;

   // - The code below is reduce the impact of setting a if-statement
   //   around queries, by setting the qid_cnt to a fixed value at this 
   //   point.
   // - mb_station_block_header will occupy one query-id.  
   #sb.z.header_qid :=
   MAX(IN1 := #mb_query.z.run.qid_cnt + 1,
       IN2 := #sb.z.header_qid);
   #mb_query.z.run.qid_cnt := #sb.z.header_qid;
END_FUNCTION

FUNCTION "mb_station_block_footer" : Void   // FC11, SCL
{ S7_Optimized_Access := 'TRUE' }
VERSION : 1.0
   VAR_IN_OUT
      sb : "mb_station_block_udt";
      mb_query : "mb_query";
   END_VAR
   VAR_TEMP
      "e" : Int;
      err : Bool;
   END_VAR
BEGIN
   // Rexhip - Extended modbus library.
   // Read the top section of mb_query for more documentation.

   REGION Recive
       IF #mb_query.z.sb.head_recive THEN
           // If there is a query that bellong to this device that has
           // recvied a resault. (with or without error)

           // Counter for exec. queries inside this station block.
           // Default is 1 query for each loop, but may be changed.
           #sb.z.exec_cnt += 1;

           // If this is the first succesfylly query after communication error,
           // then log the time this happen. (also exceptions)
           IF #sb.out.error_comm AND (
               #mb_query.stat.done
               OR #mb_query.stat.error AND NOT #mb_query.stat.error_comm)
           THEN
               #"e" := RD_LOC_T(#sb.log.connected_time);
           END_IF;

           IF #mb_query.z.sb.log_serialize_err  <> 0 THEN
               #sb.log.error_status := INT_TO_WORD(#mb_query.z.sb.log_serialize_err);
               #sb.log.error_data_addr := #mb_query.z.sb.log_data_addr;
               #sb.log.error_exception_cnt += 1;
               #sb.z.err_hold := #sb.out.error := true;

           ELSIF #mb_query.stat.error THEN // Logging - failed query        
               // Store the values for debugging. data_addr will indicate witch 
               // query caused the error, and the status is indicate the error type.
               #sb.log.error_status := #mb_query.stat.status;
               #sb.log.error_data_addr := #mb_query.z.sb.log_data_addr;

               // Two counters, one for comm.error and for all other errors.
               IF #mb_query.stat.error_comm THEN
                   #sb.log.error_comm_cnt += 1; // Eg. Bad CRC, parity, etc.
               ELSE
                   #sb.log.error_exception_cnt += 1;
               END_IF;

               // Increase communication error counter. if it's a comm.error.
               // then reset the counter.  
               IF #mb_query.stat.error_comm THEN
                   #sb.z.comm_err_cnt += BOOL_TO_USINT(#sb.z.comm_err_cnt < 255);
               ELSE
                   #sb.z.comm_err_cnt := 0;
               END_IF;

               // The error_comm flag is set if x repeating comm.errors occurres.
               #err := #sb.z.comm_err_cnt > #sb.conf.max_comm_error;
               IF #err AND NOT #sb.out.error_comm THEN
                   // Log the time when the flag is set.
                   #"e" := RD_LOC_T(#sb.log.disconnected_time);
               END_IF;
               #sb.out.error_comm := #err;

               // A comm.error will not be displayed before the
               // communication_error flag is set. Other errors will be
               // diplayed once. (NOT comm.error -> normal error)
               #sb.out.error := #sb.out.error OR NOT #mb_query.stat.error_comm
               OR #sb.out.error_comm;

               // err_hold makes the error flag stay true for more then just
               // one plc-scan.
               #sb.z.err_hold := #sb.out.error;


           ELSIF #mb_query.stat.done THEN // Logging successfully query        
               #sb.log.done_cnt += 1;
               // One successfully query -> reset 
               #sb.out.error_comm := false;
               #sb.z.comm_err_cnt := 0;
           END_IF;

           // - If it's this devices has the retry token, (sid_retry = sid_cnt)
           //   a retry has been executed and faild. Then set the retry_finished
           //   flag.
           // - The retry-token will be passed on to the next device with
           //   communication problems when the query loop has reach
           //   the end. (Inside the mb_internal_e)
           // - The library make sure that only one station block with comm.
           //   problems will do retry for each query loop revolution. 
           #mb_query.z.sb.retry_finished :=
           #mb_query.z.sb.sid_retry = #mb_query.z.sb.sid_cnt
           AND #mb_query.stat.error_comm;

           // Only one query in the SB is executed (default). The purpose is
           // to avoid a SB with many queries to occupy the bus for long periodes
           // of time. offset_qid is incread by one when a query has executed
           // given last query didn't resualt in a timeout.
           #sb.z.offset_qid += BOOL_TO_UINT(NOT #mb_query.stat.error_comm);
       END_IF;
   END_REGION

   REGION Middle
       // If all queries for this device has been executed,
       // then reset offset_qid back to the first query.
       IF #sb.z.offset_qid >
           #mb_query.z.run.qid_cnt - #sb.z.header_qid
       THEN
           #sb.z.offset_qid := 1;

           // Also reset error falg, if the last query was successfully.
           IF NOT #sb.z.err_hold THEN
               #sb.out.error := false;
           END_IF;
           #sb.z.err_hold := false;
       END_IF;

       // If the retry-token point at this device (sid_retry=sid_cnt), and there is
       // no communication problems then pass on the retry-token to the next device.
       // The retry token tell which device with communication problem that should
       // retry establish communication.
       #mb_query.z.sb.sid_retry +=
       BOOL_TO_UINT(#mb_query.z.sb.sid_retry = #mb_query.z.sb.sid_cnt
                    AND NOT #sb.out.error_comm);
   END_REGION

   REGION Finnish
       // Several condition that resault in passing on the query-token on to the
       // next device. Skipping all or the rest of the queries for this device:              
       #sb.out.finnish :=
       #mb_query.z.sb.head_recive AND ( // Skip rest of the queries if: ->
       (* *)#sb.z.exec_cnt >= #sb.conf.exec_x_quries // Some queries has executed,
       (*           *)// wait for the next loop for the remaining queries.
       (*      *)OR #mb_query.stat.error_comm) // A query resualting in comm.error    
       OR #mb_query.z.sb.head_insert AND ( // Erase a already inserted query if: ->
       (* *)#sb.out.error_comm // This station has allready comm. problems.
       (*      *)// And, it isn't this devies turn to try again.
       (*      *)AND (#mb_query.z.sb.sid_retry <> #mb_query.z.sb.sid_cnt
       (*           *)// Or, there has allready been a retry attempt on this loop.
       (*           *)OR #mb_query.z.sb.retry_finished) // (reseted in mb_internal_e)     
       (* *)OR #sb.conf.disable
       //    (* *)OR NOT #mb_query.z.sb.order // If the query isn't the next in the order
       (* *)OR #sb.conf.exec_x_quries = 0 // Zero => disable station block.
       (* *)OR #sb.conf.read_only // The read_only flag is set, and it's a write query.
       (*      *)AND #mb_query.z.run.write);

       IF #sb.out.finnish THEN // Reset
           #mb_query.z.run.insert := true;
           #mb_query.z.run.qid := #mb_query.z.run.qid_cnt + 1;
           #sb.z.exec_cnt := 0;
       END_IF;

    (*
       #mb_query.z.misc.serialize_err // Serialize or deserialize error.

       IF #mb_query.z.misc.serialize_err THEN
           //#sb.log.error_status := INT_TO_WORD(#mb_query.z.misc.serialize_err);
           #sb.log.error_data_addr := #mb_query.z.sb.recived_data_addr;
           #sb.log.error_exception_cnt += 1;
       END_IF;
      *) 
   END_REGION
END_FUNCTION

// folder: Library/Modbus/Docs

FUNCTION "mb_Debugging" : Void   // FC1, SCL
{ S7_Optimized_Access := 'TRUE' }
VERSION : 0.1
BEGIN
   (* 
   # General debugging:
   - Look online and check that the latest version of the library 
     is in use.
   - All queries need to be executed in same order, implicates from 
     the same OB.
   - Look inside the data blcok of the SB of the device that having 
     problem, and locate «#sb.log...», see if the counters are 
     running and lookup the error code of «#sb.log.error_status», 
     «#sb.log.error_data_addr» will tell witch query generating the 
     error. 

   # Modbus RTU
   - Try to increase timeout, repeaters on the bus need additional 
     time.
   - All the devies on the bus need to have a unique address.
   - Parity, buard rate, stop bits need to be the same in all 
     devices. In the modbus specification, on page 20, 19200 should be 
     default buad rate and parity should be even by default, as stated 
     on page 12. Please follow this guideline.
   - Electrical polarity. For some devices the connection "A" and "B" 
     is mislabeled, try to swap them.
   - Check for correct hardware id,

   # Modbus TCP
   - Try to increase timeout, creating a TCP-socket may take long.
   - Check IP-address.
   - Check TCP-port, 502 is default.
   - Check for unic connection-id.

   # Station Blocks (SB) creation: 
   - If mb_station_block_header has executed in one block then 
     mb_station_block_foother also need to be executed. Cheack that 
     there is no RETURN or simular between them.
   - Check datasheet of device for special requirement: function codes 
     supported, max data length, register required to be queried 
     together, etc.  
   - If the data of one query includes bools, then make sure that the 
     bools add up to whole bytes. Also make sure that all queries has 
     a length that is less then 124 words.   
   - Try to comment out sections of the queries and see if it solve 
     the problem.  

   *)
END_FUNCTION

// folder: Library/Modbus/Station blocks

FUNCTION_BLOCK "Allen_bradley_power_flex_4"   // FB16, SCL
{ S7_Optimized_Access := 'TRUE' }
VERSION : 0.1
   VAR_INPUT
      mb_addr : USInt;
      ref : Real;
      reverse : Bool;
      reset : Bool;
   END_VAR
   VAR_OUTPUT
      Output_Frequency : Real;
      Output_Current : Real;
      DC_Bus_Voltage : Real;
      Output_Voltage : Real;
   END_VAR
   VAR_IN_OUT
      mb_query : "mb_query";
   END_VAR
   VAR
      sb : "mb_station_block_udt";
      read : Struct
         stat : Struct
            x08_At_Reference : Bool;
            x09_Reference_Controlled_by_Comm : Bool;
            x10_Operation_Cmd_Controlled_by_Comm : Bool;
            x11_Parameters_have_been_locked : Bool;
            x12_Digital_Input_1_Status : Bool;
            x13_Digital_Input_2_Status : Bool;
            x14 : Bool;
            x15 : Bool;
            "x00_Ready," : Bool;
            x01_Running : Bool;
            x02_cmd_Forward : Bool;
            x03_Rotating_Forward : Bool;
            x04_Accelerating : Bool;
            "x05_Decelerating," : Bool;
            x06_Alarm : Bool;
            x07_Faulted : Bool;
         END_STRUCT;
         error_code : UInt;
         ref_feedback : UInt;
         Output_Frequency : UInt;
         Output_Current : UInt;
         DC_Bus_Voltage : UInt;
         Output_Voltage : UInt;
      END_STRUCT;
      write : Struct
         cmd : Struct
            "x08_Accel Rate 1" : Bool := TRUE;
            "x09_Accel Rate 2" : Bool;
            "x10_Decel Rate 1" : Bool := TRUE;
            "x11_Decel Rate 2" : Bool;
            x12_Freq_Source_b0 : Bool := TRUE;
            x13_Freq_Source_b1 : Bool := TRUE;
            x14_Freq_Source_b2 : Bool;
            x15 : Bool;
            x00_Stop : Bool;
            x01_Start : Bool;
            x02_Jog : Bool;
            x03_Clear_Faults : Bool;
            x04_Forward : Bool;
            x05_Reverse : Bool;
            x06 : Bool;
            x07 : Bool;
         END_STRUCT;
         ref : UInt;
      END_STRUCT;
   END_VAR
BEGIN
   // Allen Bradley - Power Flex 4 - Compact AC Drive
   //
   // http://ab.rockwellautomation.com/Drives/PowerFlex-4
   // Web: https://plc-hmi-scadas.com/gallery/PowerFlex4ModBusAddressing.pdf

   "mb_station_block_header"(sb := #sb,
                             mb_query := #mb_query);
   #mb_query.mb_addr := #mb_addr;

   #write.ref := REAL_TO_UINT(#ref * 10);
   #write.cmd.x00_Stop := #ref = 0;
   #write.cmd.x01_Start := #ref <> 0;
   #write.cmd.x03_Clear_Faults := #reset;
   #write.cmd.x04_Forward := NOT #reverse;
   #write.cmd.x05_Reverse := #reverse;

   #mb_query.mode := #mb_query.c.write.single_holding_reg;
   #mb_query(data_addr := 8192,
             data_ptr := #write.cmd);
   #mb_query(data_addr := 8193,
             data_ptr := #write.ref);

   #mb_query.mode := #mb_query.c.read.holding_reg;
   #mb_query(data_addr := 8448,
             data_ptr := #read);
   #Output_Frequency := UINT_TO_REAL(#read.Output_Frequency) / 10;
   #Output_Current := UINT_TO_REAL(#read.Output_Current) / 100;
   #DC_Bus_Voltage := UINT_TO_REAL(#read.DC_Bus_Voltage) / 10;
   #Output_Voltage := UINT_TO_REAL(#read.Output_Voltage) / 10;

   "mb_station_block_footer"(sb := #sb,
                             mb_query := #mb_query);

   (* Error codes: (read.error_codes)
   0 - No Fault
   2 - Auxilary Input
   3 - Power Loss
   4 - Undervoltage
   5 - Overvoltage
   6 - Motor Stalled
   7 - Motor Overload
   8 - Heatsink Overtemperature
   12 - HW Overcurrent (300%)
   13 - Ground Fault
   29 - Analog Input Loss
   33 - Auto Restart Tries
   38 - Phase U to Ground Short
   39 - Phase V to Ground Short
   40 - Phase W to Ground Short
   41 - Phase U/V Short
   42 - Phase U/W Short
   43 - Phase V/W Short
   63 - Software Overcurrent
   64 - Drive Overload
   70 - Power Unit Fail
   80 - AutoTune Fail
   81 - Communication Loss
   100 - Parameter Checksum Error
   122 - I/O Board Fail         
   *)
END_FUNCTION_BLOCK

FUNCTION_BLOCK "Auma_valve"   // FB17, SCL
{ S7_Optimized_Access := 'TRUE' }
VERSION : 0.1
   VAR_INPUT
      mb_addr : UInt;
   END_VAR
   VAR_IN_OUT
      mb_query : "mb_query";
   END_VAR
   VAR
      sb : "mb_station_block_udt";
      read : Struct
         status : Struct
            torque_sw_closed : Bool;
            torque_sw_open : Bool;
            limit_sw_closed : Bool;
            limit_sw_open : Bool;
            sel_sw_local : Bool;
            sel_sw_remote : Bool;
            phase_fault : Bool;
            therminal_fault : Bool;
            falt : Bool;
            warning : Bool;
            running_close : Bool;
            running_open : Bool;
            not_ready_remote : Bool;
            setpoint_reached : Bool;
            end_p_clossed : Bool;
            end_p_open : Bool;
         END_STRUCT;
         "Actual position" : UInt;
      END_STRUCT;
      write : Struct
         cmd : Struct
            byte_2 : Byte;
            open : Bool;
            close : Bool;
            use_setpoint : Bool;
            reset : Bool;
            b4 : Bool;
            b5 : Bool;
            b6 : Bool;
            b7 : Bool;
         END_STRUCT;
         setpoint : UInt;
      END_STRUCT;
   END_VAR
BEGIN
   // Auma actuator controls
   // AC 01.2/ACExC 01.2 Modbus RTU
   //
   // http://www1.auma.com/uploads/media/sp_import2/handbuecher/
   // steuerungen/hb_ac2_modbus_geraeteintegration_en.pdf

   "mb_station_block_header"(sb := #sb,
                             mb_query := #mb_query);
   #mb_query.mb_addr := #mb_addr;

   #mb_query(mode := #mb_query.c.read.input_reg,
             data_addr := 16#03E8,
             data_ptr := #read); // p.10

   #mb_query(mode := #mb_query.c.write.holding_reg,
             data_addr := 16#03E8,
             data_ptr := #write); // p.29

   "mb_station_block_footer"(sb := #sb,
                             mb_query := #mb_query);
END_FUNCTION_BLOCK

FUNCTION_BLOCK "Automatic_systems_AS1320"   // FB18, SCL
{ S7_Optimized_Access := 'TRUE' }
VERSION : 0.1
   VAR_INPUT
      mb_addr : UInt;
   END_VAR
   VAR_IN_OUT
      mb_query : "mb_query";
   END_VAR
   VAR
      sb : "mb_station_block_udt";
      read1 : Struct
         input : Word;
         input_3 : Word;
         output : Word;
         analog_in : Word;
         analog_out : Word;
         z2 : Array[1..4] of Word;
         temperature : Int;
         counter_1 : UDInt;
         counter_2 : UDInt;
         z : Array[1..3] of Word;
         state : Struct
            x08_blocked_closed : Bool;
            x09 : Bool;
            x10 : Bool;
            x11 : Bool;
            x12 : Bool;
            x13 : Bool;
            x14 : Bool;
            x15 : Bool;
            x00 : Bool;
            x01 : Bool;
            x02_open : Bool;
            x03_opening : Bool;
            x04_closed : Bool;
            x05_closing : Bool;
            x06_stop : Bool;
            x07_blocked_open : Bool;
         END_STRUCT;
      END_STRUCT;
      read2 : Struct
         PRDSTD : String[6];
         BL_xxx : String[6];
         "Type" : UInt;
         Change : UInt;
      END_STRUCT;
      write1 : Struct
         x08 : Bool;
         x09 : Bool;
         x10 : Bool;
         x11 : Bool;
         x12 : Bool;
         x13 : Bool;
         x14 : Bool;
         x15 : Bool;
         x00_open : Bool;
         x01_close : Bool;
         x02_block_open : Bool;
         x03_block_close : Bool;
         x04_stop : Bool;
         x05_reader_command_direction_a : Bool;
         x06_reader_command_direction_b : Bool;
         x07_reset_block : Bool;
      END_STRUCT;
      start_setup : Bool;
      write2 : Struct
         PS1_function : UInt;
         PS2_function : UInt;
         Positioning : UInt;
         barrier_type : UInt;
         arm_length : UInt;
         arm_type : UInt;
         power_fail_OP : UInt;
         exploitation : UInt;
      END_STRUCT;
      crank : Bool;
   END_VAR
BEGIN
   // Automatic systems - AS1320
   // http://www.visionbr.com.br/arquivo-produtos/20110823_92924_as1320-mt-en-16.pdf
   // Revision no: AS1320-prog 6.x-MT-FR-16 - 2009-11-10 

   "mb_station_block_header"(sb := #sb, mb_query := #mb_query);
   #mb_query.mb_addr := #mb_addr;

   #mb_query.mode := #mb_query.c.read.holding_reg;
   #mb_query(data_addr := 16#39, data_ptr := #read1);
   // #mb_query(data_addr := 16#00, data_ptr := #read3);
   // A micro switch at opening for the crank.
   #crank := #read1.input.%X14; 

   #mb_query.mode := #mb_query.c.write.holding_reg;
   #mb_query(data_addr := 16#12C, data_ptr := #write1);
   IF #start_setup THEN
       #mb_query(data_addr := 16#64, data_ptr := #write2);
       #start_setup := NOT #mb_query.Done;
   END_IF;

   "mb_station_block_footer"(sb := #sb, mb_query := #mb_query);
END_FUNCTION_BLOCK

FUNCTION_BLOCK "Belimo_vav_Compact_mod"   // FB19, SCL
{ S7_Optimized_Access := 'TRUE' }
VERSION : 0.1
   VAR_INPUT
      mb_addr : UInt;
      sp : Real;   // setpoint
      bus_fail_position : Real;
   END_VAR
   VAR_OUTPUT
      pos_feedback : Real;
   END_VAR
   VAR_IN_OUT
      mb_query : "mb_query";
   END_VAR
   VAR
      sb : "mb_station_block_udt";
      read : Struct
         position : Int;
      END_STRUCT;
      write1 : Struct
         setpoint : Int;
      END_STRUCT;
      write2 : Struct
         bus_fail_position : Int;
      END_STRUCT;
   END_VAR
BEGIN
   // Belimo - VAV-Compact MOD 
   // LMV-D3-MOD 5  Nm 2   W 4 VA (max. 5 A @ 5 ms) Approx. 500 g
   // NMV-D3-MOD 10 Nm 3.5 W 6 VA (max. 5 A @ 5 ms) Approx. 700 g
   // https://www.micromatic.no/globalassets/inriver/
   // resources/ko1070_0_5_1.pdf

   "mb_station_block_header"(sb := #sb, mb_query := #mb_query);
   #mb_query.mb_addr := #mb_addr;

   #mb_query.mode := #mb_query.c.read.holding_reg;
   #mb_query(data_addr := 4, data_ptr := #read);
   #pos_feedback := INT_TO_REAL(#read.position) * 0.01;

   #mb_query.mode := #mb_query.c.write.holding_reg;
   #write1.setpoint := REAL_TO_INT(#sp) * 100;
   #mb_query(data_addr := 0, data_ptr := #write1);
   #write2.bus_fail_position := REAL_TO_INT(#bus_fail_position) * 100;
   #mb_query(data_addr := 108, data_ptr := #write2);

   "mb_station_block_footer"(sb := #sb, mb_query := #mb_query);

   (*
   Bus fail position:
   0 Last setpoint (no bus monitoring)
   1 Fast close if time is exceeded
   2 Fast open if time is exceeded 
   *)
END_FUNCTION_BLOCK

FUNCTION_BLOCK "Binmaster_mnu_ultrasonic_sensor"   // FB20, SCL
{ S7_Optimized_Access := 'TRUE' }
VERSION : 0.1
   VAR_INPUT
      mb_addr : UInt;
   END_VAR
   VAR_IN_OUT
      mb_query : "mb_query";
   END_VAR
   VAR
      sb : "mb_station_block_udt";
      data : Struct
         "Model Type" : UInt;
         Raw_Distance_Level : UInt;   // [mm]
         _ : UInt;
         Temperature : Int;
         Calculated : DInt;
         __ : DWord;
         "Version" : UInt;
         "Signal Strength" : UInt;
         ___ : UInt;
         "Trip 1 Alarm" : UInt;
         "Trip 1 Status" : UInt;
         "Trip 2 Alarm" : UInt;
         "Trip 2 Status" : UInt;
      END_STRUCT;
      setting : Struct
         Units : UInt := 3;   // 3=Meters
         Distance : Struct
            Max : UInt;   // 0 - 15,250 mm
            Full : UInt;   // 0 - 15,250 mm
            Empty : UInt;
         END_STRUCT;
         cal : Struct
            Multiplier : UInt := 1000;   // 1000 -> 1.000
            Offset : UInt := 0;
         END_STRUCT;
      END_STRUCT;
   END_VAR
BEGIN
   // Binmaster - MNU Ultrasonic Sensor
   // 
   // Web: http://www.binmaster.com/_resources/e30d:ogspbx-on/files/
   // 75651567z4d4b98f5/_fn/BinMaster%20MNU%20manual%209004257%20Rev%20A1.pdf

   "mb_station_block_header"(sb := #sb, mb_query := #mb_query);
   #mb_query.mb_addr := #mb_addr;

   #mb_query.mode := #mb_query.c.mode.read;
   #mb_query(data_addr := 30299, data_ptr := #data);

   #mb_query.mode := #mb_query.c.mode.write;
   #mb_query(data_addr := 40401, data_ptr := #setting.Units);
   #mb_query(data_addr := 40405, data_ptr := #setting.Distance);
   #mb_query(data_addr := 40416, data_ptr := #setting.cal);

   "mb_station_block_footer"(sb := #sb, mb_query := #mb_query);
END_FUNCTION_BLOCK

FUNCTION_BLOCK "Danfoss_AquaDrive"   // FB21, SCL
TITLE = Danfoss AQUA-drive FC 202
{ S7_Optimized_Access := 'TRUE' }
VERSION : 0.1
   VAR_INPUT
      mb_addr : USInt;
      iRef : Real;   // s
      iStop_cost : Bool;
      iStop_ramp : Bool;
      iStop_quick : Bool;
   END_VAR
   VAR_OUTPUT
      qHz : Real;   // [hz]
      qCurrent : Real;   // [A]
      qReady : Bool;
      qRunning : Bool;
      qError : Bool;
      qIn_operation : Bool;
   END_VAR
   VAR_IN_OUT
      mb_query : "mb_query";
   END_VAR
   VAR
      sb : "mb_station_block_udt";
      serial_number : String[20];
      basic : Struct   // (unscaled)
         hz : DInt;   // x 0.1
         current : DInt;   // x 0.01
      END_STRUCT;
      stw : Struct   // Status word
         x08_Speed_eq_reference : Bool;
         x09_bus_control : Bool;
         x10_frequency_limit_ok : Bool;
         x11_in_operation : Bool;
         x12_stopped_auto_start : Bool;
         x13_voltage_exceeded : Bool;
         x14_torque_exceeded : Bool;
         x15_timer_exceeded : Bool;
         x00_control_ready : Bool;
         x01_drive_ready : Bool;
         x02_enable : Bool;   // 0=Coasting
         x03_trip : Bool;
         x04_error_no_trip : Bool;
         x05 : Bool;
         x06_triplock : Bool;
         x07_warning : Bool;
      END_STRUCT;
      ctw : Struct   // Controll word
         x08 : Bool;
         x09 : Bool;
         x10_data_valid : Bool := TRUE;
         x11 : Bool;
         x12 : Bool;
         x13 : Bool;
         x14 : Bool;
         x15_reverse : Bool;
         x00 : Bool;
         x01 : Bool;
         x02_inv_stop_ramp : Bool := TRUE;
         x03_inv_stop_coasting : Bool := TRUE;
         x04_inv_stop_quick : Bool := TRUE;
         x05_inv_hold_output_frequency : Bool := TRUE;
         x06 : Bool;
         x07_reset : Bool;
      END_STRUCT;
      state : Int;
   END_VAR
   VAR_TEMP
      "int" : Int;
      "real" : Real;
   END_VAR
BEGIN
   // Danfoss - AQUA-drive FC 202
   //
   // http://files.danfoss.com/documents/PE/doc_MG20N202.pdf
   // http://files.danfoss.com/documents/PE/doc_MG20O602.pdf 

   "mb_station_block_header"(sb := #sb, mb_query := #mb_query);
   #mb_query.mb_addr := #mb_addr;

   CASE #state OF
       0: // Action if no communication. (2=stop) 
           #"int" := 2;
           #mb_query(mode := #mb_query.c.write.holding_reg,
                     data_addr := 8039, // 8*1000+4*10-1    
                     data_ptr := #"int"); 
       1: // Select input source (2=CTW=fieldbus)
           #"int" := 2;
           #mb_query(mode := #mb_query.c.write.holding_reg,
                     data_addr := 8009, // 8*1000+1*10-1 
                     data_ptr := #"int");
       2: // Serial number 
           #mb_query(mode := #mb_query.c.read.holding_reg,
                     data_addr := 15509, // 15*1000+51*10-1
                     data_ptr := #serial_number);
   END_CASE;
   #state += BOOL_TO_INT(#mb_query.Done);
   #state := SEL(G := #state > 2 OR #sb.out.error_comm,
                 IN0 := #state, IN1 := 0);

   REGION Read 
       #mb_query.mode := #mb_query.c.read.holding_reg;
       // Status word // 16*1000+3*10-1
       #mb_query(data_addr := 16029, data_ptr := #stw);
       #qReady := #stw.x01_drive_ready AND #stw.x00_control_ready;
       #qIn_operation := #stw.x11_in_operation;
       #qError := #stw.x04_error_no_trip OR #stw.x03_trip;
       // Hz // 16*1000+13*10-1
       #mb_query(data_addr := 16129, data_ptr := #basic.hz);
       #qHz := DINT_TO_REAL(#basic.hz) * 0.1;
       // Electrical current // 16*1000+14*10-1
       #mb_query(data_addr := 16139, data_ptr := #basic.current);
       #qCurrent := DINT_TO_REAL(#basic.current) * 0.01;
       (* // RPM // 16*1000+17*10-1
       #mb_query(data_addr := 16169, data_ptr := #basic.rpm);
       #qRpm := DINT_TO_REAL(#basic.rpm) / 60; *)
   END_REGION
   REGION Write 
       #mb_query.mode := #mb_query.c.write.holding_reg;
       // CTW (controll word) // 2810 - 1 = 2809
       #ctw.x03_inv_stop_coasting := NOT #iStop_cost;
       #ctw.x02_inv_stop_ramp := NOT #iStop_ramp;
       #ctw.x04_inv_stop_quick := NOT #iStop_quick;
       #mb_query(data_addr := 2809, data_ptr := #ctw);
       // Preset reference // p.144 // 3*1000+10*10-1
       #"real" := NORM_X(MIN := 0, VALUE := #iRef, MAX := 100);
       #"int" := SCALE_X(MIN := 0, VALUE := #"real", MAX := 16#4000);
       #mb_query(data_addr := 3099, data_ptr := #"int");
   END_REGION

   "mb_station_block_footer"(sb := #sb, mb_query := #mb_query);
END_FUNCTION_BLOCK

FUNCTION_BLOCK "Delta_CFP2000"   // FB22, SCL
{ S7_Optimized_Access := 'TRUE' }
VERSION : 0.1
   VAR_INPUT
      mb_addr : USInt;
      ref : Real;   // (minus=>rev.)
   END_VAR
   VAR_OUTPUT
      stat : Struct
         drive_stops : Bool;
         drive_decelerating : Bool;
         drive_standby : Bool;
         drive_operating : Bool;
      END_STRUCT;
      current : Real;
   END_VAR
   VAR_IN_OUT
      mb_query : "mb_query";
   END_VAR
   VAR
      sb : "mb_station_block_udt";
      read : Struct
         warn_code : USInt;
         error_code : USInt;
         stat : Struct
            "b08_Master frequency controlled by communication" : Bool;
            "b09 Master frequency controlled by analog signal" : Bool;
            "b10 Operation command controlled by communication interface" : Bool;
            "b11 Parameter locked" : Bool;
            "b12 Enable to copy parameters from keypad" : Bool;
            b13 : Bool;
            b14 : Bool;
            b15 : Bool;
            b00_oper_stat : Bool;
            b01_oper_stat : Bool;
            b02 : Bool;
            b03_direction : Bool;
            b04_direction : Bool;
            b05 : Bool;
            b06 : Bool;
            b07 : Bool;
         END_STRUCT;
         frequency_cmd : Int;
         output_frequency : Int;
         output_current : UInt;
         "DC-BUS Voltage" : UInt;
         output_voltage : UInt;
         "Current step number of Multi-Step Speed Operation" : Int;
         _ : Int;
         counter_value : Int;
         power_factor_angle : Int;
         output_torque : Int;
         actual_motor_speed : Int;
         __ : Int;
         ___ : Int;
         power_output : Int;   // kwh
      END_STRUCT;
      write : Struct
         cmd_word : Struct
            b08_sel_speed : Bool;
            b09_sel_speed : Bool;
            b10_sel_speed : Bool;
            b11_sel_speed : Bool;
            b12_Enable_bit06_11_function : Bool := TRUE;
            b13_oper_keypad : Bool;
            b14_oper_Pr_00_21_setting : Bool;
            b15 : Bool;
            b00_stop : Bool;
            b01_run : Bool;
            b02 : Bool;
            b03 : Bool;
            b04_fwd : Bool;
            b05_rev : Bool;
            b06_sel_accel_decel : Bool;
            b07_sel_accel_decel : Bool;
         END_STRUCT;
         ref_freq : UInt;
         "a" : Struct
            b08 : Bool;
            b09 : Bool;
            b10 : Bool;
            b11 : Bool;
            b12 : Bool;
            b13 : Bool;
            b14 : Bool;
            b15 : Bool;
            b00_external_fault : Bool;
            b01_reset : Bool;
            b02_B_B_ON : Bool;
            b03 : Bool;
            b04 : Bool;
            b05 : Bool;
            b06 : Bool;
            b07 : Bool;
         END_STRUCT;
      END_STRUCT;
   END_VAR
BEGIN
   // Delta - CFP2000 - Variable frequency drive
   // 
   // http://www.softstartuk.com/wp-content/uploads/2017/07/VFD-CFP2000_UM_EN_20170303.pdf

   "mb_station_block_header"(sb := #sb, mb_query := #mb_query);
   #mb_query.mb_addr := #mb_addr;

   // Read
   #mb_query.mode := #mb_query.c.read.holding_reg;

   #mb_query(data_addr := 16#2100, data_ptr := #read);
   #stat.drive_stops := NOT #read.stat.b00_oper_stat AND NOT #read.stat.b01_oper_stat;
   #stat.drive_decelerating := #read.stat.b00_oper_stat AND NOT #read.stat.b01_oper_stat;
   #stat.drive_standby := NOT #read.stat.b00_oper_stat AND #read.stat.b01_oper_stat;
   #stat.drive_operating := #read.stat.b00_oper_stat AND #read.stat.b01_oper_stat;
   #current := UINT_TO_REAL(#read.output_current) * 100;
   // Output current (XX.XX A). When current is higher than
   // 655.35, it will shift decimal as (XXX.XA). The decimal
   // can refer to High byte of 211F. 

   // Write
   #mb_query.mode := #mb_query.c.write.holding_reg;

   #write.ref_freq := REAL_TO_UINT(#ref * 100);
   #write.cmd_word.b00_stop := #ref = 0;
   #write.cmd_word.b01_run := NOT #write.cmd_word.b00_stop;
   #write.cmd_word.b05_rev := #ref < 0;
   #write.cmd_word.b04_fwd := NOT #write.cmd_word.b05_rev;
   #mb_query(data_addr := 16#2000, data_ptr := #write);

   "mb_station_block_footer"(sb := #sb, mb_query := #mb_query);
END_FUNCTION_BLOCK

FUNCTION_BLOCK "Emerson_Micro_Motion"   // FB23, SCL
{ S7_Optimized_Access := 'TRUE' }
VERSION : 0.1
   VAR_INPUT
      mb_addr : UInt;
   END_VAR
   VAR_IN_OUT
      mb_query : "mb_query";
   END_VAR
   VAR
      sb : "mb_station_block_udt";
      data : Struct
         stat : Struct
            x08_Primary_mA_output_saturated : Bool;
            x09_Secondary_mA_output_saturated : Bool;
            x10_Primary_mA_output_fixed : Bool;
            x11_Secondary_mA_output_fixed : Bool;
            x12_Density_overrange : Bool;
            x13_Flowmeter_zeroing_failure : Bool;
            x14_Zero_value_too_low : Bool;
            x15_Zero_value_too_high : Bool;
            x00_EPROM_checksum_failure : Bool;
            x01_RAM_diagnostic_failure : Bool;
            x02_Sensor_failure : Bool;
            x03_Temperature_sensor_failure : Bool;
            x04_Input_overrange : Bool;
            x05_Frequency_pulse_output_saturated : Bool;
            x06_Transmitter_not_configured : Bool;
            x07_Realtime_interrupt_failure : Bool;
            x24 : Bool;
            x25 : Bool;
            x26 : Bool;
            x27 : Bool;
            x28 : Bool;
            x29 : Bool;
            x30 : Bool;
            x31 : Bool;
            x16_Transmitter_electronics_failure : Bool;
            x17_Flowmeter_zeroing_in_progress : Bool;
            x18_Slug_flow : Bool;
            x19_Power_reset_occurred : Bool;
            x20_Transmitter_configuration_changed : Bool;
            x21_Transmitter_initializing_warming_up : Bool;
            x22 : Bool;
            x23 : Bool;
         END_STRUCT;
         "Mass flow rate" : Real;
         Density : Real;
         Temperature : Real;
         "Volume flow rate" : Real;
         Pressure : Real;   // (internally derived)
         "Mass total" : Real;
         "Volume total" : Real;
         "Mass inventory" : Real;
         "Volume inventory" : Real;
      END_STRUCT;
   END_VAR
BEGIN
   // Emerson - Micro Motion Transmitters
   // RFT9739, MVD DC, Modeo 1500, Model 1700, Model 2500, Model 2700, Series 3000
   // 
   // Web: http://www2.emersonprocess.com/siteadmincenter/
   //      PM%20Micro%20Motion%20Documents/Modbus-Map-Manual-20001741.pdf

   "mb_station_block_header"(sb := #sb, mb_query := #mb_query);
   #mb_query.mb_addr := #mb_addr;

   #mb_query.mode := #mb_query.c.read.holding_reg;
   #mb_query(data_addr := 245, data_ptr := #data);

   "mb_station_block_footer"(sb := #sb, mb_query := #mb_query);
END_FUNCTION_BLOCK

FUNCTION_BLOCK "Endress_proline_promass_83"   // FB24, SCL
{ S7_Optimized_Access := 'TRUE' }
VERSION : 0.1
   VAR_INPUT
      mb_addr : UInt;
   END_VAR
   VAR_OUTPUT
      device_ok : Bool;
   END_VAR
   VAR_IN_OUT
      mb_query : "mb_query";
   END_VAR
   VAR
      sb : "mb_station_block_udt";
      data : Struct
         mass_flow : Real;
         temperature : Real;
         totalizer : Real;
         actual_system_condition : Int;   // 1->ok
      END_STRUCT;
   END_VAR
BEGIN
   // Endress - Proline Promass 83
   // Web: https://portal.endress.com/wa001/dla/5000000/5862/000/05/BA00107DEN_1311.pdf

   "mb_station_block_header"(sb := #sb, mb_query := #mb_query);
   #mb_query.mb_addr := #mb_addr;

   #mb_query(mode := #mb_query.c.read.holding_reg,
             data_addr := 5051,
             data_ptr := #data);

   "mb_station_block_footer"(sb := #sb, mb_query := #mb_query);

   #device_ok := #data.actual_system_condition = 1;
END_FUNCTION_BLOCK

FUNCTION_BLOCK "Epluse_EE071"   // FB25, SCL
{ S7_Optimized_Access := 'TRUE' }
VERSION : 0.1
   VAR_INPUT
      mb_addr : USInt := 247;
   END_VAR
   VAR_IN_OUT
      mb_query : "mb_query";
   END_VAR
   VAR
      sb : "mb_station_block_udt";
      data : Struct
         temperature_C : Real;   // [Â°C]
         temperature_F : Real;   // [Â°F]
         humidity_rel : Real;   // [%]
         humidity_abs : Real;   // [g/mÂ³]
      END_STRUCT;
      serial : String[8];
   END_VAR
BEGIN
   // Epluse - EE071
   // Humidity and Temperature Probe
   //
   // http://downloads.epluse.com/fileadmin/data/product/ee071/datasheet_EE071.pdf

   "mb_station_block_header"(sb := #sb,
                             mb_query := #mb_query);
   #mb_query.mb_addr := #mb_addr;

   #mb_query.mode := #mb_query.c.read.holding_reg;
   #mb_query(data_addr := 30026,
             data_ptr := #data);
   #mb_query(data_addr := 30001,
             data_ptr := #serial); // 30001-30008

   "mb_station_block_footer"(sb := #sb,
                             mb_query := #mb_query);

   IF #sb.out.error_comm THEN
       #data.temperature_C := 0;
       #data.temperature_F := 0;
       #data.humidity_rel := 0;
       #data.humidity_abs := 0;
   END_IF;

   (* Electrical connections

   Supply voltage 1) 2) 4 - 28 V DC

   brown...+UB
   white.....B-RS485 (= Data-)
   blue......A-RS485 (= Data+)
   black....GND
   grey......shielding

   1...+UB
   2...B-RS485 (= Data-)
   3...A-RS485 (= Data+)
   4...GND

   *)
END_FUNCTION_BLOCK

FUNCTION_BLOCK "G_Instruments_GpH141_MB"   // FB26, SCL
{ S7_Optimized_Access := 'TRUE' }
VERSION : 0.1
   VAR_INPUT
      mb_addr : USInt;
   END_VAR
   VAR_OUTPUT
      voltage_mV : Real;
      pH : Real;
      temperature : Real;
   END_VAR
   VAR_IN_OUT
      mb_query : "mb_query";
   END_VAR
   VAR
      sb : "mb_station_block_udt";
      change_mb_addr : Struct
         old : UInt;
         new : UInt;
      END_STRUCT;
   END_VAR
   VAR_TEMP
      read1 : Struct
         voltage : Int;
         pH : Int;   // compensated for temperature
         temperature : Int;
      END_STRUCT;
   END_VAR
BEGIN
   // G Instruments - GpH141-MB - pH/ORP Transmitter
   // Part number: 30535.
   // http://www.ginstruments.com/files/GpH141-MB.pdf

   "mb_station_block_header"(sb := #sb,
                             mb_query := #mb_query);
   #mb_query.mb_addr := #mb_addr;

   #mb_query.mode := #mb_query.c.read.holding_reg;

   #mb_query(data_addr := 19,
             data_ptr := #read1);
   IF #mb_query.Done THEN
       #voltage_mV := INT_TO_REAL(#read1.voltage) / 10;
       #pH := INT_TO_REAL(#read1.pH) / 100;
       #temperature := INT_TO_REAL(#read1.temperature) / 10;
   END_IF;

   (* IF #change_mb_addr.new <> 0 AND #change_mb_addr.old <> 0 THEN
       #mb_query(mb_addr := #change_mb_addr.old,
                 mode := #mb_query.c.write.single_holding_reg,
                 data_addr := 1200,
                 data_ptr := #change_mb_addr.new);
       IF #mb_query.Done THEN #change_mb_addr.new := 0; END_IF;
   END_IF; *)

   "mb_station_block_footer"(sb := #sb,
                             mb_query := #mb_query);

   (*
   Default comm. setting: 19200 bps, even parity, addr 1.

   Electrical connection:
   10 is A (D+)
   11 is RS485 ground (isolated from all other grounds)
   12 is B (D-)
   *)
END_FUNCTION_BLOCK

FUNCTION_BLOCK "hitachi_wj200_series"   // FB27, SCL
{ S7_Optimized_Access := 'TRUE' }
VERSION : 0.1
   VAR_INPUT
      mb_addr : USInt;
      ref : Real;
      acceleration_time : Real := 30.0;   // sec
      deceleration_time : Real := 30.0;   // sec
   END_VAR
   VAR_OUTPUT
      output_frequency : Real;
      output_current : Real;
   END_VAR
   VAR_IN_OUT
      mb_query : "mb_query";
   END_VAR
   VAR
      sb : "mb_station_block_udt";
      save_param : Bool;
      read1 : Struct
         output_frequency : UDInt;   // 0.01 [Hz]
         output_current : UInt;   // 0.1 [A]
         rotation_direction : Int;   // 0: Stopping, 1: Forward, 2:Reverse
      END_STRUCT;
      read2 : Struct
         torque : Int;   // [%]
         output_voltage : UInt;   // 0.1 [V]
         output_power : UInt;   // 0.1 [kW]
         watt_hour : UDInt;   // 0.1 [wh]
         elapsed_run_time : UDInt;   // [h]
         elapsed_power_on_time : UDInt;   // [h]
         "heat sink_temperature" : UDInt;   // 0.1 [℃]
      END_STRUCT;
      read3_Life_check : Struct
         x08 : Bool;
         x09 : Bool;
         x10 : Bool;
         x11 : Bool;
         x12 : Bool;
         x13 : Bool;
         x14 : Bool;
         x15 : Bool;
         x00_Capacitor_on_main_circuit_board : Bool;
         x01_cooling_fan : Bool;
         x02 : Bool;
         x03 : Bool;
         x04 : Bool;
         x05 : Bool;
         x06 : Bool;
         x07 : Bool;
      END_STRUCT;
      read4_Ambient_temperature : Int;
      read5_trip : Struct
         cnt : UInt;
         info : Array[1..3] of Struct
            factor : UInt;
            status : UInt;
            frequency : DInt;
            current : UInt;
            voltage : UInt;
            running_time : UDInt;   // [h] Cumulative running time at tripping
            powerOn_time : UDInt;   // [h] Cumulative power-on time at tripping
         END_STRUCT;
      END_STRUCT;
      read6_status : Struct
         "A" : UInt;
         "B" : UInt;   // 0: Stopping, 1: Running, 2: Tripping
         C : UInt;
      END_STRUCT;
      read7 : Struct
         x0_inverter_ready : Bool;
         x1_forward : Bool;
         x2_reverse : Bool;
         x3_major_failure : Bool;
         x4_data_writing_in_progress : Bool;
         x5 : Bool;
         x6 : Bool;
         x7 : Bool;
      END_STRUCT;
      write1 : Struct
         acceleration_time_1 : UDInt := 3000;   // x0.01 sec
         deceleration_time_1 : UDInt := 3000;   // x0.01 sec
      END_STRUCT;
      write2_source : Struct
         frequency_source : UInt := 3;   // 3:Modbus
         run_command_source : UInt := 3;   // 3:Modbus
      END_STRUCT;
      write3_comm_error : Struct
         communication_watchdog_timer : UInt := 1000;   // 0.01 [sec.]
         communication_error_action : UInt := 4;
      END_STRUCT;
      write5 : Struct
         x0_Run : Bool;
         x1_Reverse : Bool;
         x2_Trip : Bool;
         x3_Reset : Bool;
         x4 : Bool;
         x5 : Bool;
         x6 : Bool;
         x7 : Bool;
      END_STRUCT;
      write6_DC_breaking : Struct
         enable : UInt;   // 0 (disabling), 1 (enabling), 2 (output freq < [A052])
         frequency : UInt;   // 0.01 [Hz]
         wait_time : UInt;   // 0.1 [sec.]
         force_during_deceleration : UInt;   // [%]
         time_for_deceleration : UInt;   // 0.1 [sec.]
      END_STRUCT;
   END_VAR
   VAR_TEMP
      tmp : Word;
      write4_frequency : DInt;   // 0.01 [Hz]
   END_VAR
BEGIN
   // Hitachi WJ200-series
   // Manual Number: NT325X
   // https://www.hitachi-america.us/supportingdocs/forbus/inverters/Support/WJ200_Instruction_NT325X.pdf

   "mb_station_block_header"(sb := #sb, mb_query := #mb_query);
   #mb_query.mb_addr := #mb_addr;

   // --- Read queries
   #mb_query.mode := #mb_query.c.read.holding_reg;
   #mb_query(data_addr := 16#1001, data_ptr := #read1);
   #mb_query(data_addr := 16#1010, data_ptr := #read2);
   #mb_query(data_addr := 16#101d, data_ptr := #read3_Life_check);
   #mb_query(data_addr := 16#134e, data_ptr := #read4_Ambient_temperature);
   #mb_query(data_addr := 16#0011, data_ptr := #read5_trip);
   #mb_query(data_addr := 16#0003, data_ptr := #read6_status);

   #output_frequency := UDINT_TO_REAL(#read1.output_frequency) / 100;
   #output_current := UINT_TO_REAL(#read1.output_current) / 10;

   #mb_query(mode := #mb_query.c.read.discrete_output,
             data_addr := 16#0045,
             data_ptr := #read7);

   // --- Write queries ---
   #write4_frequency := REAL_TO_DINT(#ref * 100);
   #write1.acceleration_time_1 := REAL_TO_UDINT(#acceleration_time * 100);
   #write1.deceleration_time_1 := REAL_TO_UDINT(#deceleration_time * 100);

   #mb_query.mode := #mb_query.c.write.holding_reg;
   #mb_query(data_addr := 16#1103, data_ptr := #write1);
   #mb_query(data_addr := 16#1201, data_ptr := #write2_source);
   #mb_query(data_addr := 16#162e, data_ptr := #write3_comm_error);
   #mb_query(data_addr := 16#0001, data_ptr := #write4_frequency);
   #mb_query(data_addr := 16#1245, data_ptr := #write6_DC_breaking);

   // Save data to EEPROM. 
   IF #save_param THEN
       #mb_query(mode := #mb_query.c.write.single_holding_reg,
                 data_addr := 16#0900,
                 data_ptr := #tmp);
       #save_param := NOT #mb_query.Done;
   END_IF;

   #write5.x0_Run := #ref <> 0;
   #mb_query(mode := #mb_query.c.write.discrete_output,
             data_addr := 16#0001,
             data_len := 4,
             data_ptr := #write5);

   #mb_query.data_len := #mb_query.c.auto_len;
   "mb_station_block_footer"(sb := #sb, mb_query := #mb_query);

   (*
   === read6_status ===
   .A
   0: Initial status
   2: Stopping
   3: Running
   4: Free-run stop
   5: Jogging
   6: DC braking
   7: Retrying
   8: Tripping
   9: Undervoltage (UV), 

   .C
   1: Stopping
   2: Decelerating
   3: Constant-speed operation
   4: Accelerating
   5: Forward rotation
   6: Reverse rotation
   7: Switching from fwd. to rev. rotation,
   8: Switching from rev. to fwd. rotation,
   9: Starting fwd.
   10: Starting rev

   === write3_comm_error.communication_error_action === 
   0 (tripping), 
   1 (tripping after decelerating and stopping the motor), 
   2 (ignoring errors),
   3 (stopping the motor after free-running),
   4 (decelerating and stopping the motor) 

   === Save data to EEPROM === 
   The service life of the storage element of the inverter is 
   limited to about 100,000 write operations.  Frequent use of 
   the ENTER command may shorten its service life.

   === read5_trip.info ===
   .factor: 
   00 No trip factor 0 
   01 Over-current event while at constant speed 1 
   02 Over-current event during deceleration 2 
   03 Over-current event during acceleration 3 
   04 Over-current event during other conditions 4 
   05 Overload protection 5 
   06 Braking resistor overload protection 6 
   07 Overvoltage protection 7 
   08 EEPROM error 8 
   09 Undervoltage protection 9
   10 Current detection error 10
   11 CPU error 11
   12 External trip 12
   13 USP error 13
   14 Ground-fault protection 14
   15 Input overvoltage protection 15
   21 Inverter thermal trip 21
   22 CPU error 22
   25 Main circuit error 25
   30 Driver error 30
   35 Thermistor error 35
   36 Braking error 36
   37 Safe Stop 37
   38 Low-speed overload protection 38
   40 Operator connection 40
   41 Modbus communication error 41
   43 Easy sequence error (invalid instruction) 43
   44 Easy sequence error (invalid nesting count) 44
   45 Easy sequence execution error 1 45
   50 Easy sequence user trip 0 to 9, 50 to 59
   60 Option error 0 to 9, 60 to 69
   80 Encoder disconnection 80
   81 Excessive speed 81
   83 Position control range trip 83

   .status
   0: Resetting 
   1: Stopping 
   2: Decelerating 
   3: Constant-speed operation 
   4: Accelerating 
   5: Operating at zero frequency 
   6: Starting 
   7: DC braking 
   8: Overload restricted 

   *)
END_FUNCTION_BLOCK

FUNCTION_BLOCK "InSitu_RDO_PRO_X"   // FB30, SCL
{ S7_Optimized_Access := 'TRUE' }
VERSION : 0.1
   VAR_INPUT
      mb_addr : UInt;
   END_VAR
   VAR_OUTPUT
      dissolved_oxygen : Real;   // mg/L
      temperature : Real;   // C
      saturation : Real;   // %
      oxygen_partial_pressure : Real;   // mbar
      alarm : Bool;
   END_VAR
   VAR_IN_OUT
      mb_query : "mb_query";
   END_VAR
   VAR
      sb : "mb_station_block_udt";
      read1 : Array[1..4] of Struct
         value : Real;
         Parameter_ID : UInt;
         Units_ID : UInt;
         data_quality : UInt;
         "Off line_sentinel_value" : UInt;
         Available_Units : UInt;
      END_STRUCT;
      read2 : Struct
         serial_number : UDInt;
         manufacture_date : Array[1..3] of UInt;
      END_STRUCT;
      device_name : String[32];
   END_VAR
   VAR_TEMP
      tmp_alarm : Bool;
      c : Int;
   END_VAR
BEGIN
   // InSitu - RDO PRO X
   // 
   // https://in-situ.com/wp-content/uploads/2015/08/
   // RDO_PRO-X_-Titan_Modbus_SDI-12-_Guide.pdf

   "mb_station_block_header"(sb := #sb, mb_query := #mb_query);
   #mb_query.mb_addr := #mb_addr;

   #mb_query.mode := #mb_query.c.read.holding_reg;
   #mb_query(data_addr := 38, data_ptr := #read1);
   #mb_query(data_addr := 9002, data_ptr := #read2);
   #mb_query(data_addr := 9019, data_ptr := #device_name);

   #dissolved_oxygen := #read1[1].value;
   #temperature := #read1[2].value;
   #saturation := #read1[3].value;
   #oxygen_partial_pressure := #read1[4].value;
   FOR #c := 1 TO 4 DO
       #tmp_alarm := #tmp_alarm OR #read1[#c].data_quality <> 0;
   END_FOR;
   #alarm := #tmp_alarm;

   "mb_station_block_footer"(sb := #sb, mb_query := #mb_query);

   (* 
   === Sensor health table: ===
   0  Normal Data Quality
   1  Parameter measured without errors using an expired user 
      calibration. (User Cal Expired)
   2  Parameter measured without errors using an expired factory 
      calibration. (Factory Cal Expired)
   3  Parameter measured with error, sentinel value supplied. 
   4  Sensor is warming up, sentinel value supplied.
   5  Parameter measured but does not meet normal quality 
      criteria. The sensor has sustained moderate damage, or  
      the recommended lifespan has been reached.
   *)
END_FUNCTION_BLOCK

